Staubli VAL3: IO.pjx

--- IO.pjx ---
Parameters version=s7.7 stackSize=5000 millimeterUnit=true
Program file=Action.pgx
Program file=ActionLCF.pgx
Program file=Alarm.pgx
Program file=AtHome.pgx
Program file=AtHomePulse.pgx
Program file=Axis7Action.pgx
Program file=Axis7onPosition.pgx
Program file=Axis7OnReady.pgx
Program file=Axis7Status.pgx
Program file=Axis8Action.pgx
Program file=Axis8onPosition.pgx
Program file=Axis8OnReady.pgx
Program file=Axis8Status.pgx
Program file=AxisDoor.pgx
Program file=AxisIsNeg.pgx
Program file=AxisJogSpeed.pgx
Program file=AxisTest.pgx
Program file=CanProduct.pgx
Program file=ChoosehansPro.pgx
Program file=ChooseMultPro.pgx
Program file=CloseWeld.pgx
Program file=Digtal2Analog.pgx
Program file=Digtal2AnalogS.pgx
Program file=ExtraContrAxis.pgx
Program file=GasChoose.pgx
Program file=GetAxis7Pos.pgx
Program file=GetAxis8Pos.pgx
Program file=GetAxisStatus.pgx
Program file=GetKeyIO.pgx
Program file=GetPreset.pgx
Program file=Init.pgx
Program file=IOName.pgx
Program file=IOvalue.pgx
Program file=IsDigtal.pgx
Program file=IsInput.pgx
Program file=KeyDigtalIO.pgx
Program file=Light.pgx
Program file=MatchSpdPreset.pgx
Program file=PerforatiAction.pgx
Program file=Preset.pgx
Program file=PresetLaser.pgx
Program file=ProductPoll.pgx
Program file=ProductReady.pgx
Program file=ReadMe.pgx
Program file=SafteyIO.pgx
Program file=SendSpeed.pgx
Program file=start.pgx
Program file=stop.pgx
Program file=TrajBypass.pgx
Program file=WaitProIOEnd.pgx
Program file=WeldAction.pgx
Program file=WeldProgChoose.pgx
Program file=WorkPlaceFinish.pgx
Data file=IO.dtx

--- IO.dtx ---
public aio aAio{}
  [In4_a7CurPosH] = {link=ModbusSrv-0\Modbus-Word\In4_a7CurPosH}
  [In4_a7CurPosL] = {link=ModbusSrv-0\Modbus-Word\In4_a7CurPosL}
  [In4_a8CurPosH] = {link=ModbusSrv-0\Modbus-Word\In4_a8CurPosH}
  [In4_a8CurPosL] = {link=ModbusSrv-0\Modbus-Word\In4_a8CurPosL}
  [In_aVersion] = {link=ModbusSrv-0\Modbus-Word\In_aVersion}
  [O1_aAirPress] = {link=ModbusSrv-0\Modbus-Word\O1_aAirPress}
  [O1_aFPWM] = {link=ModbusSrv-0\Modbus-Word\O1_aFPWM}
  [O1_aLasPwr] = {link=ModbusSrv-0\Modbus-Word\O1_aLasPwr}
  [O1_aPMW] = {link=ModbusSrv-0\Modbus-Word\O1_aPMW}
  [O2_aFollowSensitive] = {link=ModbusSrv-0\Modbus-Word\O2_aFollowSensitive}
  [O2_aNull] = {link=ModbusSrv-0\Modbus-Word\O2_aNull}
  [O4_a7AiHomeH] = {link=ModbusSrv-0\Modbus-Word\O4_a7AiHomeH}
  [O4_a7AiHomeL] = {link=ModbusSrv-0\Modbus-Word\O4_a7AiHomeL}
  [O4_a7JogVelo] = {link=ModbusSrv-0\Modbus-Word\O4_a7JogVelo}
  [O4_a7MoveDis] = {link=ModbusSrv-0\Modbus-Word\O4_a7MoveDis}
  [O4_a7MovePosH] = {link=ModbusSrv-0\Modbus-Word\O4_a7MovePosH}
  [O4_a7MovePosL] = {link=ModbusSrv-0\Modbus-Word\O4_a7MovePosL}
  [O4_a7Velocity] = {link=ModbusSrv-0\Modbus-Word\O4_a7Velocity}
  [O4_a8AiHomeH] = {link=ModbusSrv-0\Modbus-Word\O4_a8AiHomeH}
  [O4_a8AiHomeL] = {link=ModbusSrv-0\Modbus-Word\O4_a8AiHomeL}
  [O4_a8JogVelo] = {link=ModbusSrv-0\Modbus-Word\O4_a8JogVelo}
  [O4_a8MoveDis] = {link=ModbusSrv-0\Modbus-Word\O4_a8MoveDis}
  [O4_a8MovePosH] = {link=ModbusSrv-0\Modbus-Word\O4_a8MovePosH}
  [O4_a8MovePosL] = {link=ModbusSrv-0\Modbus-Word\O4_a8MovePosL}
  [O4_a8Velocity] = {link=ModbusSrv-0\Modbus-Word\O4_a8Velocity}
  [Out_a114_129] = {link=ModbusSrv-0\Modbus-Word\Out_a114_129}
  [Out_a130_133] = {link=ModbusSrv-0\Modbus-Word\Out_a130_133}
  [Out_a66_81] = {link=ModbusSrv-0\Modbus-Word\Out_a66_81}
  [Out_a82_97] = {link=ModbusSrv-0\Modbus-Word\Out_a82_97}
  [Out_a98_113] = {link=ModbusSrv-0\Modbus-Word\Out_a98_113}
public bool bAxisDoorEnable
bool bDigFollowHight
public bool bDigtal[167]
  [0] = true
  [1] = true
  [2] = true
  [3] = true
  [4] = true
  [5] = true
  [6] = true
  [7] = true
  [8] = true
  [9] = true
  [10] = true
  [11] = true
  [12] = true
  [13] = true
  [14] = true
  [15] = true
  [16] = true
  [17] = true
  [18] = true
  [19] = true
  [20] = true
  [21] = true
  [22] = true
  [23] = true
  [24] = true
  [25] = true
  [26] = true
  [27] = true
  [28] = true
  [29] = true
  [30] = true
  [31] = true
  [32] = true
  [33] = true
  [34] = true
  [35] = true
  [36] = true
  [37] = true
  [38] = true
  [39] = true
  [40] = true
  [41] = true
  [42] = true
  [43] = true
  [44] = true
  [45] = true
  [46] = true
  [47] = true
  [48] = true
  [49] = true
  [50] = true
  [51] = true
  [52] = true
  [53] = true
  [54] = true
  [55] = true
  [56] = true
  [57] = true
  [58] = true
  [59] = true
  [60] = true
  [61] = true
  [62] = true
  [63] = true
  [64] = true
  [65] = true
  [66] = true
  [67] = true
  [68] = true
  [69] = true
  [70] = true
  [71] = true
  [72] = true
  [73] = true
  [74] = true
  [75] = true
  [76] = true
  [77] = true
  [78] = true
  [79] = true
  [80] = true
  [81] = true
  [82] = true
  [83] = true
  [84] = true
  [85] = true
  [86] = true
  [87] = true
  [88] = true
  [89] = true
  [90] = true
  [91] = true
  [92] = true
  [93] = true
  [94] = true
  [95] = true
  [96] = true
  [97] = true
  [98] = true
  [99] = true
  [100] = true
  [101] = true
  [102] = true
  [103] = true
  [104] = true
  [105] = true
  [106] = true
  [107] = true
  [108] = true
  [109] = true
  [110] = true
  [111] = true
  [112] = true
  [113] = true
  [114] = true
  [115] = true
  [116] = true
  [117] = true
  [118] = true
  [119] = true
  [120] = true
  [121] = true
  [122] = true
  [123] = true
  [124] = true
  [125] = true
  [126] = true
  [127] = true
  [128] = true
  [129] = true
  [130] = true
  [131] = true
  [132] = true
  [133] = true
  [134] = true
public bool bExt7AxisEnable
public bool bExt8AxisEnable
public bool bGunUp
bool bWaitActionOff
bool bWaitFollowDown
public bool bWeldEnable
public dio dDio{}
  [In1_bEndCycl] = {link=ModbusSrv-0\Modbus-Bit\In1_bEndCycl}
  [In1_bHome] = {link=ModbusSrv-0\Modbus-Bit\In1_bHome}
  [In1_bNull1] = {link=ModbusSrv-0\Modbus-Bit\In1_bNull1}
  [In1_bNull2] = {link=ModbusSrv-0\Modbus-Bit\In1_bNull2}
  [In1_bNull3] = {link=ModbusSrv-0\Modbus-Bit\In1_bNull3}
  [In1_bOutAlarm] = {link=ModbusSrv-0\Modbus-Bit\In1_bOutAlarm}
  [In1_bPausCycl] = {link=ModbusSrv-0\Modbus-Bit\In1_bPausCycl}
  [In1_bPeripheralReady] = {link=ModbusSrv-0\Modbus-Bit\In1_bPeripheralReady}
  [In1_bPowerOn] = {link=ModbusSrv-0\Modbus-Bit\In1_bPowerOn}
  [In1_bPrdSta1] = {link=ModbusSrv-0\Modbus-Bit\In1_bPrdSta1}
  [In1_bPrdSta2] = {link=ModbusSrv-0\Modbus-Bit\In1_bPrdSta2}
  [In1_bReset] = {link=ModbusSrv-0\Modbus-Bit\In1_bReset}
  [In1_bStartCycl] = {link=ModbusSrv-0\Modbus-Bit\In1_bStartCycl}
  [In1_bStopCycl] = {link=ModbusSrv-0\Modbus-Bit\In1_bStopCycl}
  [In2_bAirAlarm] = {link=ModbusSrv-0\Modbus-Bit\In2_bAirAlarm}
  [In2_bCollisonAlarm] = {link=ModbusSrv-0\Modbus-Bit\In2_bCollisonAlarm}
  [In2_bContactAlarm] = {link=ModbusSrv-0\Modbus-Bit\In2_bContactAlarm}
  [In2_bLaserAlarm] = {link=ModbusSrv-0\Modbus-Bit\In2_bLaserAlarm}
  [In2_bNull1] = {link=ModbusSrv-0\Modbus-Bit\In2_bNull1}
  [In2_bNull2] = {link=ModbusSrv-0\Modbus-Bit\In2_bNull2}
  [In2_bNull3] = {link=ModbusSrv-0\Modbus-Bit\In2_bNull3}
  [In2_bNull4] = {link=ModbusSrv-0\Modbus-Bit\In2_bNull4}
  [In2_bNull5] = {link=ModbusSrv-0\Modbus-Bit\In2_bNull5}
  [In2_bNull6] = {link=ModbusSrv-0\Modbus-Bit\In2_bNull6}
  [In2_bNull7] = {link=ModbusSrv-0\Modbus-Bit\In2_bNull7}
  [In2_bNull8] = {link=ModbusSrv-0\Modbus-Bit\In2_bNull8}
  [In2_bNull9] = {link=ModbusSrv-0\Modbus-Bit\In2_bNull9}
  [In2_bPrdSta3] = {link=ModbusSrv-0\Modbus-Bit\In2_bPrdSta3}
  [In2_bPrdSta4] = {link=ModbusSrv-0\Modbus-Bit\In2_bPrdSta4}
  [In2_bRasterOn] = {link=ModbusSrv-0\Modbus-Bit\In2_bRasterOn}
  [In4_b7BackHome] = {link=ModbusSrv-0\Modbus-Bit\In4_b7BackHome}
  [In4_b7HomeDone] = {link=ModbusSrv-0\Modbus-Bit\In4_b7HomeDone}
  [In4_b7IsHome] = {link=ModbusSrv-0\Modbus-Bit\In4_b7IsHome}
  [In4_b7MotorError] = {link=ModbusSrv-0\Modbus-Bit\In4_b7MotorError}
  [In4_b7MotorPower] = {link=ModbusSrv-0\Modbus-Bit\In4_b7MotorPower}
  [In4_b7Reached] = {link=ModbusSrv-0\Modbus-Bit\In4_b7Reached}
  [In4_b8BackHome] = {link=ModbusSrv-0\Modbus-Bit\In4_b8BackHome}
  [In4_b8HomeDone] = {link=ModbusSrv-0\Modbus-Bit\In4_b8HomeDone}
  [In4_b8IsHome] = {link=ModbusSrv-0\Modbus-Bit\In4_b8IsHome}
  [In4_b8MotorError] = {link=ModbusSrv-0\Modbus-Bit\In4_b8MotorError}
  [In4_b8MotorPower] = {link=ModbusSrv-0\Modbus-Bit\In4_b8MotorPower}
  [In4_b8Reached] = {link=ModbusSrv-0\Modbus-Bit\In4_b8Reached}
  [In4_bNull1] = {link=ModbusSrv-0\Modbus-Bit\In4_bNull1}
  [In4_bNull2] = {link=ModbusSrv-0\Modbus-Bit\In4_bNull2}
  [In4_bNull3] = {link=ModbusSrv-0\Modbus-Bit\In4_bNull3}
  [In4_bNull4] = {link=ModbusSrv-0\Modbus-Bit\In4_bNull4}
  [In4_bNull5] = {link=ModbusSrv-0\Modbus-Bit\In4_bNull5}
  [In4_bNull6] = {link=ModbusSrv-0\Modbus-Bit\In4_bNull6}
  [In4_bNull7] = {link=ModbusSrv-0\Modbus-Bit\In4_bNull7}
  [In4_bNull8] = {link=ModbusSrv-0\Modbus-Bit\In4_bNull8}
  [In7_bDownLimit_7] = {link=ModbusSrv-0\Modbus-Bit\In7_bDownLimit_7}
  [In7_bHomeLimit_7] = {link=ModbusSrv-0\Modbus-Bit\In7_bHomeLimit_7}
  [In7_bNull1] = {link=ModbusSrv-0\Modbus-Bit\In7_bNull1}
  [In7_bUpLimit_7] = {link=ModbusSrv-0\Modbus-Bit\In7_bUpLimit_7}
  [In8_bDownLimit_8] = {link=ModbusSrv-0\Modbus-Bit\In8_bDownLimit_8}
  [In8_bHomeLimit_8] = {link=ModbusSrv-0\Modbus-Bit\In8_bHomeLimit_8}
  [In8_bNull1] = {link=ModbusSrv-0\Modbus-Bit\In8_bNull1}
  [In8_bUpLimit_8] = {link=ModbusSrv-0\Modbus-Bit\In8_bUpLimit_8}
  [O1_bAirOn] = {link=ModbusSrv-0\Modbus-Bit\O1_bAirOn}
  [O1_bAlarm] = {link=ModbusSrv-0\Modbus-Bit\O1_bAlarm}
  [O1_bFollowDone] = {link=ModbusSrv-0\Modbus-Bit\O1_bFollowDone}
  [O1_bFollowOn] = {link=ModbusSrv-0\Modbus-Bit\O1_bFollowOn}
  [O1_bGreenLamp] = {link=ModbusSrv-0\Modbus-Bit\O1_bGreenLamp}
  [O1_bLaserOn] = {link=ModbusSrv-0\Modbus-Bit\O1_bLaserOn}
  [O1_bNull1] = {link=ModbusSrv-0\Modbus-Bit\O1_bNull1}
  [O1_bRedLamp] = {link=ModbusSrv-0\Modbus-Bit\O1_bRedLamp}
  [O1_bYellowLamp] = {link=ModbusSrv-0\Modbus-Bit\O1_bYellowLamp}
  [O2_bAxisPos1] = {link=ModbusSrv-0\Modbus-Bit\O2_bAxisPos1}
  [O2_bAxisPos2] = {link=ModbusSrv-0\Modbus-Bit\O2_bAxisPos2}
  [O2_bAxisPos3] = {link=ModbusSrv-0\Modbus-Bit\O2_bAxisPos3}
  [O2_bFollowHeigh1] = {link=ModbusSrv-0\Modbus-Bit\O2_bFollowHeigh1}
  [O2_bFollowHeigh2] = {link=ModbusSrv-0\Modbus-Bit\O2_bFollowHeigh2}
  [O2_bFollowHeigh3] = {link=ModbusSrv-0\Modbus-Bit\O2_bFollowHeigh3}
  [O2_bNull1] = {link=ModbusSrv-0\Modbus-Bit\O2_bNull1}
  [O2_bNull2] = {link=ModbusSrv-0\Modbus-Bit\O2_bNull2}
  [O2_bNull3] = {link=ModbusSrv-0\Modbus-Bit\O2_bNull3}
  [O2_bProCode1] = {link=ModbusSrv-0\Modbus-Bit\O2_bProCode1}
  [O2_bProCode2] = {link=ModbusSrv-0\Modbus-Bit\O2_bProCode2}
  [O2_bProCode3] = {link=ModbusSrv-0\Modbus-Bit\O2_bProCode3}
  [O2_bSta1Stat] = {link=ModbusSrv-0\Modbus-Bit\O2_bSta1Stat}
  [O2_bSta2Stat] = {link=ModbusSrv-0\Modbus-Bit\O2_bSta2Stat}
  [O2_bSta3Stat] = {link=ModbusSrv-0\Modbus-Bit\O2_bSta3Stat}
  [O2_bSta4Stat] = {link=ModbusSrv-0\Modbus-Bit\O2_bSta4Stat}
  [O4_b7AxisHome] = {link=ModbusSrv-0\Modbus-Bit\O4_b7AxisHome}
  [O4_b7ChkHome] = {link=ModbusSrv-0\Modbus-Bit\O4_b7ChkHome}
  [O4_b7MoveDir] = {link=ModbusSrv-0\Modbus-Bit\O4_b7MoveDir}
  [O4_b7MoveDirM] = {link=ModbusSrv-0\Modbus-Bit\O4_b7MoveDirM}
  [O4_b7MoveToPos] = {link=ModbusSrv-0\Modbus-Bit\O4_b7MoveToPos}
  [O4_b7RecordPos] = {link=ModbusSrv-0\Modbus-Bit\O4_b7RecordPos}
  [O4_b7ResetError] = {link=ModbusSrv-0\Modbus-Bit\O4_b7ResetError}
  [O4_b7StopMotor] = {link=ModbusSrv-0\Modbus-Bit\O4_b7StopMotor}
  [O4_b8AxisHome] = {link=ModbusSrv-0\Modbus-Bit\O4_b8AxisHome}
  [O4_b8ChkHome] = {link=ModbusSrv-0\Modbus-Bit\O4_b8ChkHome}
  [O4_b8MoveDir] = {link=ModbusSrv-0\Modbus-Bit\O4_b8MoveDir}
  [O4_b8MoveDirM] = {link=ModbusSrv-0\Modbus-Bit\O4_b8MoveDirM}
  [O4_b8MoveToPos] = {link=ModbusSrv-0\Modbus-Bit\O4_b8MoveToPos}
  [O4_b8RecordPos] = {link=ModbusSrv-0\Modbus-Bit\O4_b8RecordPos}
  [O4_b8ResetError] = {link=ModbusSrv-0\Modbus-Bit\O4_b8ResetError}
  [O4_b8StopMotor] = {link=ModbusSrv-0\Modbus-Bit\O4_b8StopMotor}
  [O4_bHome] = {link=ModbusSrv-0\Modbus-Bit\O4_bHome}
  [O4_bNull1] = {link=ModbusSrv-0\Modbus-Bit\O4_bNull1}
  [O4_bNull2] = {link=ModbusSrv-0\Modbus-Bit\O4_bNull2}
  [O4_bNull3] = {link=ModbusSrv-0\Modbus-Bit\O4_bNull3}
  [O4_bNull4] = {link=ModbusSrv-0\Modbus-Bit\O4_bNull4}
  [O4_bNull5] = {link=ModbusSrv-0\Modbus-Bit\O4_bNull5}
  [O4_bNull6] = {link=ModbusSrv-0\Modbus-Bit\O4_bNull6}
  [O4_bNull7] = {link=ModbusSrv-0\Modbus-Bit\O4_bNull7}
  [O4_bNull8] = {link=ModbusSrv-0\Modbus-Bit\O4_bNull8}
  [O7_bAxis7Direction] = {link=ModbusSrv-0\Modbus-Bit\O7_bAxis7Direction}
  [O7_bAxis7Pulse] = {link=ModbusSrv-0\Modbus-Bit\O7_bAxis7Pulse}
  [O7_bNull1] = {link=ModbusSrv-0\Modbus-Bit\O7_bNull1}
  [O7_bNull2] = {link=ModbusSrv-0\Modbus-Bit\O7_bNull2}
  [O7_bNull3] = {link=ModbusSrv-0\Modbus-Bit\O7_bNull3}
  [O8_bAxis8Direction] = {link=ModbusSrv-0\Modbus-Bit\O8_bAxis8Direction}
  [O8_bAxis8Pulse] = {link=ModbusSrv-0\Modbus-Bit\O8_bAxis8Pulse}
  [O8_bNull1] = {link=ModbusSrv-0\Modbus-Bit\O8_bNull1}
  [O8_bNull2] = {link=ModbusSrv-0\Modbus-Bit\O8_bNull2}
  [O8_bNull3] = {link=ModbusSrv-0\Modbus-Bit\O8_bNull3}
  [UsIn_bNull1] = {link=ModbusSrv-0\Modbus-Bit\UsIn_bNull1}
  [UsIn_bNull2] = {link=ModbusSrv-0\Modbus-Bit\UsIn_bNull2}
  [UsIn_bNull3] = {link=ModbusSrv-0\Modbus-Bit\UsIn_bNull3}
  [UsIn_bNull4] = {link=ModbusSrv-0\Modbus-Bit\UsIn_bNull4}
  [UsIn_bNull5] = {link=ModbusSrv-0\Modbus-Bit\UsIn_bNull5}
  [UsIn_bNull6] = {link=ModbusSrv-0\Modbus-Bit\UsIn_bNull6}
  [UsIn_bNull7] = {link=ModbusSrv-0\Modbus-Bit\UsIn_bNull7}
  [UsIn_bNull8] = {link=ModbusSrv-0\Modbus-Bit\UsIn_bNull8}
  [UsO_bNull1] = {link=ModbusSrv-0\Modbus-Bit\UsO_bNull1}
  [UsO_bNull2] = {link=ModbusSrv-0\Modbus-Bit\UsO_bNull2}
  [UsO_bNull3] = {link=ModbusSrv-0\Modbus-Bit\UsO_bNull3}
  [UsO_bNull4] = {link=ModbusSrv-0\Modbus-Bit\UsO_bNull4}
  [UsO_bNull5] = {link=ModbusSrv-0\Modbus-Bit\UsO_bNull5}
  [UsO_bNull6] = {link=ModbusSrv-0\Modbus-Bit\UsO_bNull6}
  [UsO_bNull7] = {link=ModbusSrv-0\Modbus-Bit\UsO_bNull7}
  [UsO_bNull8] = {link=ModbusSrv-0\Modbus-Bit\UsO_bNull8}
public string sIOName[167]
  [0] = "无"
  [1] = "In1_bPowerOn"
  [2] = "In1_bStartCycl"
  [3] = "In1_bStopCycl"
  [4] = "In1_bHome"
  [5] = "In1_bEndCycl"
  [6] = "In1_bPrdSta1"
  [7] = "In1_bPrdSta2"
  [8] = "In1_bPausCycl"
  [9] = "In1_bOutAlarm"
  [10] = "In1_bReset"
  [11] = "In1_bPeripheralReady"
  [12] = "In1_bNull1"
  [13] = "In1_bNull2"
  [14] = "In1_bNull3"
  [15] = "UsIn_bNull1"
  [16] = "UsIn_bNull2"
  [17] = "UsIn_bNull3"
  [18] = "UsIn_bNull4"
  [19] = "UsIn_bNull5"
  [20] = "UsIn_bNull6"
  [21] = "UsIn_bNull7"
  [22] = "UsIn_bNull8"
  [23] = "In2_bPrdSta3"
  [24] = "In2_bPrdSta4"
  [25] = "In2_bAirAlarm"
  [26] = "In2_bCollisonAlarm"
  [27] = "In2_bLaserAlarm"
  [28] = "In2_bContactAlarm"
  [29] = "In2_bRasterOn"
  [30] = "In2_bNull1"
  [31] = "In2_bNull2"
  [32] = "In2_bNull3"
  [33] = "In2_bNull4"
  [34] = "In2_bNull5"
  [35] = "In2_bNull6"
  [36] = "In2_bNull7"
  [37] = "In2_bNull8"
  [38] = "In2_bNull9"
  [39] = "In7_bUpLimit_7"
  [40] = "In7_bDownLimit_7"
  [41] = "In7_bHomeLimit_7"
  [42] = "In7_bNull1"
  [43] = "In8_bUpLimit_8"
  [44] = "In8_bDownLimit_8"
  [45] = "In8_bHomeLimit_8"
  [46] = "In8_bNull1"
  [47] = "In4_b7Reached"
  [48] = "In4_b7BackHome"
  [49] = "In4_b7HomeDone"
  [50] = "In4_b7MotorPower"
  [51] = "In4_b7IsHome"
  [52] = "In4_b7MotorError"
  [53] = "In4_b8Reached"
  [54] = "In4_b8BackHome"
  [55] = "In4_b8HomeDone"
  [56] = "In4_b8MotorPower"
  [57] = "In4_b8IsHome"
  [58] = "In4_b8MotorError"
  [59] = "In4_bNull1"
  [60] = "In4_bNull2"
  [61] = "In4_bNull3"
  [62] = "In4_bNull4"
  [63] = "In4_bNull5"
  [64] = "In4_bNull6"
  [65] = "In4_bNull7"
  [66] = "In4_bNull8"
  [67] = "O1_bLaserOn"
  [68] = "O1_bFollowOn"
  [69] = "O1_bFollowDone"
  [70] = "O1_bAirOn"
  [71] = "O1_bNull1"
  [72] = "O1_bRedLamp"
  [73] = "O1_bYellowLamp"
  [74] = "O1_bGreenLamp"
  [75] = "O1_bAlarm"
  [76] = "UsO_bNull1"
  [77] = "UsO_bNull2"
  [78] = "UsO_bNull3"
  [79] = "UsO_bNull4"
  [80] = "UsO_bNull5"
  [81] = "UsO_bNull6"
  [82] = "UsO_bNull7"
  [83] = "UsO_bNull8"
  [84] = "O2_bSta1Stat"
  [85] = "O2_bSta2Stat"
  [86] = "O2_bSta3Stat"
  [87] = "O2_bSta4Stat"
  [88] = "O2_bProCode1"
  [89] = "O2_bProCode2"
  [90] = "O2_bProCode3"
  [91] = "O2_bFollowHeigh1"
  [92] = "O2_bFollowHeigh2"
  [93] = "O2_bFollowHeigh3"
  [94] = "O2_bAxisPos1"
  [95] = "O2_bAxisPos2"
  [96] = "O2_bAxisPos3"
  [97] = "O2_bNull1"
  [98] = "O2_bNull2"
  [99] = "O2_bNull3"
  [100] = "O7_bAxis7Pulse"
  [101] = "O7_bAxis7Direction"
  [102] = "O7_bNull1"
  [103] = "O7_bNull2"
  [104] = "O7_bNull3"
  [105] = "O8_bAxis8Pulse"
  [106] = "O8_bAxis8Direction"
  [107] = "O8_bNull1"
  [108] = "O8_bNull2"
  [109] = "O8_bNull3"
  [110] = "O4_b7RecordPos"
  [111] = "O4_b7MoveToPos"
  [112] = "O4_b7ResetError"
  [113] = "O4_b7ChkHome"
  [114] = "O4_b7AxisHome"
  [115] = "O4_b7MoveDir"
  [116] = "O4_b7MoveDirM"
  [117] = "O4_b7StopMotor"
  [118] = "O4_bHome"
  [119] = "O4_b8RecordPos"
  [120] = "O4_b8MoveToPos"
  [121] = "O4_b8ResetError"
  [122] = "O4_b8ChkHome"
  [123] = "O4_b8AxisHome"
  [124] = "O4_b8MoveDir"
  [125] = "O4_b8MoveDirM"
  [126] = "O4_b8StopMotor"
  [127] = "O4_bNull1"
  [128] = "O4_bNull2"
  [129] = "O4_bNull3"
  [130] = "O4_bNull4"
  [131] = "O4_bNull5"
  [132] = "O4_bNull6"
  [133] = "O4_bNull7"
  [134] = "O4_bNull8"
  [135] = "O1_aLasPwr"
  [136] = "O1_aAirPress"
  [137] = "O1_aFPWM"
  [138] = "O1_aPMW"
  [139] = "O2_aFollowSensitive"
  [140] = "O2_aNull"
  [141] = "In4_a7CurPosL"
  [142] = "In4_a7CurPosH"
  [143] = "In4_a8CurPosL"
  [144] = "In4_a8CurPosH"
  [145] = "O4_a7Velocity"
  [146] = "O4_a7JogVelo"
  [147] = "O4_a7MoveDis"
  [148] = "O4_a7AiHomeH"
  [149] = "O4_a7AiHomeL"
  [150] = "O4_a7MovePosL"
  [151] = "O4_a7MovePosH"
  [152] = "O4_a8Velocity"
  [153] = "O4_a8JogVelo"
  [154] = "O4_a8MoveDis"
  [155] = "O4_a8AiHomeH"
  [156] = "O4_a8AiHomeL"
  [157] = "O4_a8MovePosL"
  [158] = "O4_a8MovePosH"
  [159] = "Out_a66_81"
  [160] = "Out_a82_97"
  [161] = "Out_a98_113"
  [162] = "Out_a114_129"
  [163] = "Out_a130_133"
  [164] = "In_aVersion"
  [165] = "延时"
  [166] = "收弧时间"
public bool bUserIOReset

--- IO123.dtx ---
mdesc mNomSpeed
public string sIOName
public bool bDigtal

--- start.pgx ---
public program start()
begin
  //所有的IO动作都要写入log文件中
  //信号一般作为脉冲信号来处理
  //



  call Init()

  while true


    call Digtal2Analog()
    delay(0)
  endWhile
end

--- Action.pgx ---
public program Action(num& x_nAction[] (dimensions=2), bool x_bMoveId, num x_nMoveID)
  local bool l_bFirst
  local bool l_bInput
  local bool l_bNull
  local num l_nLast
  local num l_nNum
begin
  //延时是否需要停止等待？
  //




  //一共是每个点上最多12个IO


  //如果都为空，则直接跳出
  l_bNull=false
  for l_nNum=0 to 11
    l_bNull=x_nAction[l_nNum,0]!=0 or x_nAction[l_nNum,1]!=0 or l_bNull
  endFor
  if !l_bNull
    return
  endIf




  //通过MOVEID来实现
  for l_nNum=0 to 11

    //如果后面的都是0则退出
    l_bNull=false
    for l_nLast=l_nNum to 11
      l_bNull=x_nAction[l_nLast,0]!=0 or x_nAction[l_nLast,1]!=0 or l_bNull
    endFor
    if !l_bNull
      return
    endIf


    //通过MOVEID来实现
    if x_bMoveId
      call IsInput(x_nAction[l_nNum,0],l_bInput)
      //如果有等待信号，直接退出
      if l_bInput
        return
      else
        wait(getMoveId()>x_nMoveID+0.8)
        call IOvalue(x_nAction[l_nNum,0],x_nAction[l_nNum,1])
      endIf





     //
    else

      //跟在运动指令后面
      call IsInput(x_nAction[l_nNum,0],l_bInput)
      //如果有等待信号 则运行
      if l_bInput
        l_bFirst=true

      endIf

      if l_bFirst
        //如果不是收弧时间


        if x_nAction[l_nNum,0]!=166 and l_bInput
          if x_nMoveID==-2
            waitEndMove()
          else
            if x_nMoveID>=0
              wait(getMoveId()>x_nMoveID+0.8)
            endIf
          endIf
        endIf
      endIf

      call IOvalue(x_nAction[l_nNum,0],x_nAction[l_nNum,1])


      if x_nAction[l_nNum,0]==166
        //  logMsg(toString(".3",x_nAction[l_nNum,1]))
        logMsg(toString(".3",clock())+"  "+toString(".3",getMoveId()))
      endIf


    endIf


    //把数字量输出
    call Digtal2Analog()

  endFor


end

--- ActionLCF.pgx ---
public program ActionLCF(num& x_nAction[] (dimensions=2), bool x_bMoveId, num x_nMoveID, num x_nActionBuff)
  local bool l_bFirst
  local bool l_bInput
  local bool l_bNull
  local num l_nLast
  local num l_nNum
begin
  //2016.01.26
  //特定为激光融覆定制的程序



  //延时是否需要停止等待？
  //

  x_nActionBuff=max(0.01,min(0.8,x_nActionBuff))


  //一共是每个点上最多12个IO


  //如果都为空，则直接跳出
  l_bNull=false
  for l_nNum=0 to 11
    l_bNull=x_nAction[l_nNum,0]!=0 or x_nAction[l_nNum,1]!=0 or l_bNull
  endFor
  if !l_bNull
    return
  endIf




  //通过MOVEID来实现
  for l_nNum=0 to 11

    //如果后面的都是0则退出
    l_bNull=false
    for l_nLast=l_nNum to 11
      l_bNull=x_nAction[l_nLast,0]!=0 or x_nAction[l_nLast,1]!=0 or l_bNull
    endFor
    if !l_bNull
      return
    endIf


    //通过MOVEID来实现
    if x_bMoveId
      call IsInput(x_nAction[l_nNum,0],l_bInput)
      //如果有等待信号，直接退出
      if l_bInput
        return
      else
        wait(getMoveId()>x_nMoveID+x_nActionBuff)
        call IOvalue(x_nAction[l_nNum,0],x_nAction[l_nNum,1])
      endIf





     //
    else

      //跟在运动指令后面
      call IsInput(x_nAction[l_nNum,0],l_bInput)
      //如果有等待信号 则运行
      if l_bInput
        l_bFirst=true

      endIf

      if l_bFirst
        //如果不是收弧时间


        if x_nAction[l_nNum,0]!=166 and l_bInput
          if x_nMoveID==-2
            waitEndMove()
          else
            if x_nMoveID>=0
              wait(getMoveId()>x_nMoveID+x_nActionBuff)
            endIf
          endIf
        endIf
      endIf

      call IOvalue(x_nAction[l_nNum,0],x_nAction[l_nNum,1])


      if x_nAction[l_nNum,0]==166
        //  logMsg(toString(".3",x_nAction[l_nNum,1]))
        logMsg(toString(".3",clock())+"  "+toString(".3",getMoveId()))
      endIf


    endIf


    //把数字量输出
    call Digtal2Analog()

  endFor


end

--- Alarm.pgx ---
public program Alarm(num x_nDelay (dimensions=1), num x_nInterface (dimensions=1), bool& x_bAlarm (dimensions=1))
  local bool l_bEstop
  local string l_sS
begin
  //外设报警信号触发

  //外部綜合报警，七轴报警，八轴报警
  //碰撞报警，气体报警，随动报警


  x_bAlarm=false
  call IOName(9,l_sS)
  x_bAlarm=(x_bAlarm or dDio[l_sS]==true)
  call IOName(25,l_sS)
  x_bAlarm=(x_bAlarm or dDio[l_sS]==true)
  call IOName(26,l_sS)
  x_bAlarm=(x_bAlarm or dDio[l_sS]==true)
  call IOName(27,l_sS)
  x_bAlarm=(x_bAlarm or dDio[l_sS]==true)
  call IOName(28,l_sS)
  x_bAlarm=(x_bAlarm or dDio[l_sS]==true)

  //外部七轴报警
  if bExt7AxisEnable
    call IOName(52,l_sS)
    x_bAlarm=(x_bAlarm or dDio[l_sS]==true)
  endIf

  //外部八轴报警
  if bExt8AxisEnable
    call IOName(58,l_sS)
    x_bAlarm=(x_bAlarm or dDio[l_sS]==true)
  endIf

  delay(0)
  //急停按钮输入
  l_bEstop=esStatus()==2
  dDio["O1_bAlarm"]=l_bEstop
  x_bAlarm=(l_bEstop or x_bAlarm)

  //报警或者机器人没有上电，则会停止外部轴运动
  if x_bAlarm or !isPowered()
    if dDio["O4_b7StopMotor"]==false
      dDio["O4_b7StopMotor"]=true
    endIf
    if dDio["O4_b8StopMotor"]==false
      dDio["O4_b8StopMotor"]=true
    endIf
  endIf


  //如果再次确认报警
  if x_bAlarm

    //如果机器人在上电状态，再次确认
    if isPowered()
      delay(min(max(0,x_nDelay),5))
      //再次确认
      x_bAlarm=false
      call IOName(9,l_sS)
      x_bAlarm=(dDio[l_sS]==true or x_bAlarm)
      call IOName(25,l_sS)
      x_bAlarm=(dDio[l_sS]==true or x_bAlarm)
      call IOName(26,l_sS)
      x_bAlarm=(dDio[l_sS]==true or x_bAlarm)
      call IOName(27,l_sS)
      x_bAlarm=(dDio[l_sS]==true or x_bAlarm)
      call IOName(28,l_sS)
      x_bAlarm=(dDio[l_sS]==true or x_bAlarm)

      //外部七轴
      if bExt7AxisEnable
        call IOName(52,l_sS)
        x_bAlarm=(dDio[l_sS]==true or x_bAlarm)
      endIf

      //外部八轴
      if bExt8AxisEnable
        call IOName(58,l_sS)
        x_bAlarm=(dDio[l_sS]==true or x_bAlarm)
      endIf

    endIf

    //查看机器人是否报警
    if x_bAlarm
      call Light(0)
      if isPowered()
        disablePower()
        //        logMsg("Modbus IO输入报警触发")
        call IOName(9,l_sS)
        if dDio[l_sS]==true
          popUpMsg("In1_bOutAlarm  外部综合报警触发")
          logMsg("In1_bOutAlarm  外部综合报警触发")
        endIf


        call IOName(25,l_sS)
        if dDio[l_sS]==true
          popUpMsg("In2_bAirAlarm  气体报警触发")
          logMsg("In2_bAirAlarm  气体报警触发")
        endIf

        call IOName(26,l_sS)
        if dDio[l_sS]==true
          popUpMsg("In2_bCollisonAlarm  碰撞报警触发")
          logMsg("In2_bCollisonAlarm  碰撞报警触发")
        endIf

        call IOName(27,l_sS)
        if dDio[l_sS]==true
          popUpMsg("In2_bLaserAlarm  激光报警触发")
          logMsg("In2_bLaserAlarm  激光报警触发")
        endIf

        call IOName(28,l_sS)
        if dDio[l_sS]==true
          popUpMsg("In2_bContactAlarm  触碰报警触发")
          logMsg("In2_bContactAlarm  触碰报警触发")
        endIf

        call IOName(52,l_sS)
        if dDio[l_sS]==true
          popUpMsg("In4_b7MotorError 七轴报警触发")
          logMsg("In4_b7MotorError 七轴报警触发")
        endIf

        call IOName(58,l_sS)
        if dDio[l_sS]==true
          popUpMsg("In4_b8MotorError  八轴报警触发")
          logMsg("In4_b8MotorError  八轴报警触发")
        endIf

      endIf
      call KeyDigtalIO(false,false,false,0,0)
      //      call SafteyIO(false)
      //      call SafteyIO(true)
    endIf

  else
    if x_nInterface!=13
      call Light(1)
    endIf
  endIf

end

--- AtHome.pgx ---
public program AtHome(bool x_bHome (dimensions=1))
begin


  dDio["O1_bFollowDone"]=x_bHome
  call Digtal2Analog()







end

--- AtHomePulse.pgx ---
public program AtHomePulse()
begin

  //2014.12.09
  //回零脉冲
  waitEndMove()
  dDio["UsO_bNull2"]=true
  call Digtal2Analog()
  delay(0.5)
  dDio["UsO_bNull2"]=false
  call Digtal2Analog()


  //信号确认
  delay(0.5)
  dDio["UsO_bNull1"]=true
  delay(0.5)
  dDio["UsO_bNull1"]=false
  delay(0.5)
  dDio["UsO_bNull7"]=true
  delay(0.5)
  dDio["UsO_bNull7"]=false
  delay(0.5)


end

--- Axis7Action.pgx ---
public program Axis7Action(num x_nType (dimensions=1))
begin

  //七轴的IO动作

  switch x_nType

    //点动正
    case 1
      if dDio["O4_b7StopMotor"]==true
        dDio["O4_b7StopMotor"]=false
        delay(0.05)
      endIf
      dDio["O4_b7MoveDir"]=true
      // aioSet(aAio["O4_a7JogVelo"],50)
      delay(0.2)

    break


    //点动负
    case 2
      if dDio["O4_b7StopMotor"]==true
        dDio["O4_b7StopMotor"]=false
        delay(0.05)
      endIf

      dDio["O4_b7MoveDirM"]=true
      //  aioSet(aAio["O4_a7JogVelo"],50)
      delay(0.2)
    break

    //回到机械零位
    case 4
      dDio["O4_b7StopMotor"]=false
      dDio["O4_b7AxisHome"]=true
      delay(0.2)
    break





    //停止运动
    case 6
      dDio["O4_b7StopMotor"]=true
      delay(0.2)
      dDio["O4_b7StopMotor"]=false
    break




    //没有按钮按下
    case 9
      dDio["O4_b7ResetError"]=false
      dDio["O4_b7AxisHome"]=false
      dDio["O4_b7MoveDirM"]=false
      dDio["O4_b7MoveDir"]=false
    break


    //复位
    case 10
      dDio["O4_b7StopMotor"]=false
      dDio["O4_b7ResetError"]=true
      delay(0.2)
      // dDio["O4_b7ResetError"]=false
    break
    default
    break

  endSwitch


end

--- Axis7onPosition.pgx ---
public program Axis7onPosition(num x_nPos (dimensions=1), num x_nPrecent (dimensions=1), bool& x_bOK (dimensions=1))
  local num l_nNum
begin

  x_bOK=false
  call GetAxis7Pos(l_nNum,x_nPrecent)
  x_bOK=abs(l_nNum-x_nPos)<0.001

end

--- Axis7OnReady.pgx ---
public program Axis7OnReady(num x_nPosition (dimensions=1), num x_nSpeed (dimensions=1), num x_nPrecent (dimensions=1), bool& x_bRes (dimensions=1))
  local bool l_bBool
  local num l_nNum
begin

  //异步七轴运动到位


  x_bRes=false

  //参数合法性
  if x_nSpeed<=0 or x_nPrecent<=0 or x_nPosition<=0
    return
  endIf


  //没有电或者报警
  if dDio["In4_b7MotorPower"]==false or dDio["In4_b7MotorError"]==true or dDio["In4_b7BackHome"]==false
    return
  endIf

  call AxisIsNeg(false,l_bBool)
  if l_bBool
    return
  endIf


  dDio["O4_b7RecordPos"]=true
  delay(0.2)
  dDio["O4_b7RecordPos"]=false

  call GetAxis7Pos(l_nNum,x_nPrecent)
  if abs(l_nNum-x_nPosition)!=0
    waitEndMove()
  else
    x_bRes=true
    return
  endIf
  dDio["O4_b7StopMotor"]=false
  delay(0.2)
  x_nPosition=x_nPosition*x_nPrecent
  aioSet(aAio["O4_a7Velocity"],max(1,x_nSpeed*x_nPrecent*16.666667))
  aioSet(aAio["O4_a7MovePosL"],x_nPosition%power(2,16))
  aioSet(aAio["O4_a7MovePosH"],roundDown(x_nPosition/power(2,16)))
  dDio["O4_b7MoveToPos"]=true
  delay(0.2)
  dDio["O4_b7MoveToPos"]=false

  x_nPosition=x_nPosition/x_nPrecent
  while dDio["In4_b7Reached"]!=true or abs(l_nNum-x_nPosition)>10
    call GetAxis7Pos(l_nNum,x_nPrecent)
    if dDio["O4_b7StopMotor"]==true
      x_bRes=false
      return
    endIf
    delay(0)
  endWhile

  x_bRes=true



end

--- Axis7Status.pgx ---
public program Axis7Status(bool& x_bPowerOn (dimensions=1), bool& x_bAlarm (dimensions=1), bool& x_bhome (dimensions=1))
begin

  //  x_bAlarm=true
  //  x_bPowerOn=false

  x_bhome=dDio["In4_b7BackHome"]==true
  x_bPowerOn=dDio["In4_b7MotorPower"]==true
  x_bAlarm=dDio["In4_b7MotorError"]==true











end

--- Axis8Action.pgx ---
public program Axis8Action(num x_nType (dimensions=1))
begin

  //七轴的IO动作

  switch x_nType

    //点动正
    case 1
      if dDio["O4_b8StopMotor"]==true
        dDio["O4_b8StopMotor"]=false
        delay(0.05)
      endIf
      dDio["O4_b8MoveDir"]=true
      //aioSet(aAio["O4_a8JogVelo"],50)
      delay(0.2)

    break

    //点动负
    case 2
      if dDio["O4_b8StopMotor"]==true
        dDio["O4_b8StopMotor"]=false
        delay(0.05)
      endIf
      dDio["O4_b8MoveDirM"]=true
      //  aioSet(aAio["O4_a8JogVelo"],50)
      delay(0.2)
    break

    //回到机械零位
    case 4
      dDio["O4_b8StopMotor"]=false
      dDio["O4_b8AxisHome"]=true
      delay(0.2)
    break





    //停止运动
    case 6
      dDio["O4_b8StopMotor"]=true
      delay(0.2)
      dDio["O4_b8StopMotor"]=false
    break


    case 6

    break


    //没有按钮按下
    case 9
      dDio["O4_b8ResetError"]=false
      dDio["O4_b8AxisHome"]=false
      dDio["O4_b8MoveDirM"]=false
      dDio["O4_b8MoveDir"]=false
    break


    //复位
    case 10
      dDio["O4_b8StopMotor"]=false
      dDio["O4_b8ResetError"]=true
      // dDio["O4_b8StopMotor"]=false
      delay(0.2)
    break
    default
    break

  endSwitch


end

--- Axis8onPosition.pgx ---
public program Axis8onPosition(num x_nPos (dimensions=1), num x_nPrecent (dimensions=1), bool& x_bOK (dimensions=1))
  local num l_nNum
begin

  x_bOK=false
  call GetAxis8Pos(l_nNum,x_nPrecent)
  x_bOK=abs(l_nNum-x_nPos)<0.001

end

--- Axis8OnReady.pgx ---
public program Axis8OnReady(num x_nPosition (dimensions=1), num x_nSpeed (dimensions=1), num x_nPrecent (dimensions=1), bool& x_bRes (dimensions=1))
  local bool l_bBool
  local num l_nNum
begin


  //异步八轴到位
  x_bRes=false

  //参数合法性
  if x_nSpeed<=0 or x_nPrecent<=0 or x_nPosition<=0
    return
  endIf



  //没有电或者报警
  if dDio["In4_b8MotorPower"]==false or dDio["In4_b8MotorError"]==true or dDio["In4_b8BackHome"]==false
    return
  endIf

  call AxisIsNeg(true,l_bBool)
  if l_bBool
    return
  endIf


  dDio["O4_b8RecordPos"]=true
  delay(0.2)
  dDio["O4_b8RecordPos"]=false

  call GetAxis8Pos(l_nNum,x_nPrecent)

  if abs(l_nNum-x_nPosition)!=0
    waitEndMove()
  else
    x_bRes=true
    return
  endIf

  dDio["O4_b8StopMotor"]=false
  delay(0.2)
  x_nPosition=x_nPosition*x_nPrecent
  aioSet(aAio["O4_a8Velocity"],max(1,x_nSpeed*x_nPrecent*16.666667))
  aioSet(aAio["O4_a8MovePosL"],x_nPosition%power(2,16))
  aioSet(aAio["O4_a8MovePosH"],roundDown(x_nPosition/power(2,16)))
  dDio["O4_b8MoveToPos"]=true
  delay(0.2)
  dDio["O4_b8MoveToPos"]=false

  x_nPosition=x_nPosition/x_nPrecent
  while dDio["In4_b8Reached"]!=true or abs(l_nNum-x_nPosition)>10
    call GetAxis8Pos(l_nNum,x_nPrecent)
    if dDio["O4_b8StopMotor"]==true
      x_bRes=false
      return
    endIf
    delay(0)
  endWhile

  x_bRes=true


end

--- Axis8Status.pgx ---
public program Axis8Status(bool& x_bPowerOn (dimensions=1), bool& x_bAlarm (dimensions=1), bool& x_bhome (dimensions=1))
begin
  //  x_bAlarm=true
  //  x_bPowerOn=false
  x_bhome=dDio["In4_b8BackHome"]==true
  x_bPowerOn=dDio["In4_b8MotorPower"]==true
  x_bAlarm=dDio["In4_b8MotorError"]==true


end

--- AxisDoor.pgx ---
public program AxisDoor(bool x_bOpen (dimensions=1), bool x_b8Axis (dimensions=1))
begin
  //门开关信号
  //为外部轴七轴和八轴进行打开安全门使用
  //法利莱
  //安全门信号设置


  //如果门打不开，则打不开
  if !bAxisDoorEnable
    return
  endIf


  //x_bOpen   true 打开门   false 门关闭
  //x_b8Axis  true  八轴    false 七轴


  //七八轴打开
  if !x_b8Axis
    //七轴打开
    if x_bOpen
      dDio["UsO_bNull5"]=true
      wait(dDio["UsIn_bNull5"]==true and dDio["UsIn_bNull6"]==false)
    else
      dDio["UsO_bNull5"]=false
      wait(dDio["UsIn_bNull6"]==true and dDio["UsIn_bNull5"]==false)

    endIf


  else
    //八轴打开
    if x_bOpen
      dDio["UsO_bNull6"]=true
      wait(dDio["UsIn_bNull7"]==true and dDio["UsIn_bNull8"]==false)
    else
      dDio["UsO_bNull6"]=false
      wait(dDio["UsIn_bNull8"]==true and dDio["UsIn_bNull7"]==false)

    endIf
  endIf



end

--- AxisIsNeg.pgx ---
public program AxisIsNeg(bool x_b8Axis (dimensions=1), bool& x_bRes (dimensions=1))
begin
  x_bRes=false

  if x_b8Axis
    x_bRes=aioGet(aAio["In4_a8CurPosH"])>=3000

  else

    x_bRes=aioGet(aAio["In4_a7CurPosH"])>=3000

  endIf





end

--- AxisJogSpeed.pgx ---
public program AxisJogSpeed(num x_nSpeed, bool x_b8Axis)
begin

  //修改点动速度
  //修改1这个是比例系数

  x_nSpeed=max(0,min(100,x_nSpeed))
  if x_b8Axis

    aioSet(aAio["O4_a8JogVelo"],x_nSpeed*1)

  else
    aioSet(aAio["O4_a7JogVelo"],x_nSpeed*1)

  endIf




end

--- AxisTest.pgx ---
public program AxisTest()
begin
  dDio["O1_bFollowOn"]=true
  delay(0.5)
  dDio["O1_bFollowOn"]=false
  delay(0.5)
  dDio["O1_bFollowOn"]=true
  delay(0.5)
  dDio["O1_bFollowOn"]=false
  delay(0.5)


end

--- CanProduct.pgx ---
public program CanProduct(num& x_nWorkPlace (dimensions=1))
begin
  //等待IO响应



  //第一工位
  if dDio["In1_bPrdSta1"]==true
    delay(0.2)
    if watch(dDio["In1_bPrdSta1"]==true,0.1)
      if watch(dDio["In1_bPrdSta1"]==false,2)
        logMsg("In1_bPrdSta1触发:工位1信号被触发")
        //      x_bCanProuct[1]=true
        x_nWorkPlace=1
        return
      endIf
    endIf
  endIf

  //第二工位
  if dDio["In1_bPrdSta2"]==true
    delay(0.2)
    if watch(dDio["In1_bPrdSta2"]==true,0.1)
      if watch(dDio["In1_bPrdSta2"]==false,2)
        logMsg("In1_bPrdSta2触发:工位2信号被触发")
        //x_bCanProuct[2]=true
        x_nWorkPlace=2
        return
      endIf
    endIf
  endIf


  //第三工位
  if dDio["In2_bPrdSta3"]==true
    delay(0.2)
    if watch(dDio["In2_bPrdSta3"]==true,0.1)
      if watch(dDio["In2_bPrdSta3"]==false,2)
        logMsg("In2_bPrdSta3触发:工位3信号被触发")
        //      x_bCanProuct[3]=true
        x_nWorkPlace=3
        return
      endIf
    endIf
  endIf

  //第四工位
  if dDio["In2_bPrdSta4"]==true
    delay(0.2)
    if watch(dDio["In2_bPrdSta4"]==true,0.1)
      //      x_bCanProuct[4]=true
      if watch(dDio["In2_bPrdSta4"]==false,2)
        logMsg("In2_bPrdSta4触发:工位4信号被触发")
        x_nWorkPlace=4
        return
      endIf
    endIf
  endIf



end

--- ChoosehansPro.pgx ---
public program ChoosehansPro(num& x_nWorkPlace (dimensions=1), num& x_nProductIndex (dimensions=1), num& x_nMax[] (dimensions=1))
  local num l_nNum
begin
  //  //2013.10.30
  //  //通过数字量来选择产品
  //  //主要用来检测按钮触发
  //  //同工位多产品函数

  //2014.05.30





  //  x_nProductIndex=0
  //  x_nProductIndex=0
  //  l_nNum=0

  if x_nProductIndex>=x_nMax[x_nWorkPlace]
    x_nProductIndex=0
  endIf

  if x_nProductIndex>0
    x_nProductIndex=x_nProductIndex+1
    return

  endIf

  while true
    //工位1
    if dDio["In1_bPrdSta1"]==true and dDio["UsIn_bNull1"]==true and dDio["UsIn_bNull2"]==true
      delay(0.1)
      if dDio["In1_bPrdSta1"]==true and dDio["UsIn_bNull1"]==true and dDio["UsIn_bNull2"]==true
        //
        x_nProductIndex=1
        x_nWorkPlace=1
        return
      endIf
    endIf


    //工位2
    if dDio["In1_bPrdSta2"]==true and dDio["UsIn_bNull3"]==true and dDio["UsIn_bNull3"]==true
      delay(0.1)
      if dDio["In1_bPrdSta2"]==true and dDio["UsIn_bNull3"]==true and dDio["UsIn_bNull4"]==true
        //
        x_nProductIndex=1
        x_nWorkPlace=2
        return
      endIf
    endIf


    //工位3
    if dDio["In1_bPrdSta2"]==true and dDio["UsIn_bNull5"]==true and dDio["UsIn_bNull6"]==true
      delay(0.1)
      if dDio["In1_bPrdSta2"]==true and dDio["UsIn_bNull5"]==true and dDio["UsIn_bNull6"]==true
        //
        x_nProductIndex=1
        x_nWorkPlace=3
        return
      endIf
    endIf







    //2014.06.03
    //*************************************************************************
    //*************************************************************************

    //为大族定制
    //A1,A2,A3,A4
    if dDio["In1_bPrdSta1"]==true and dDio["UsIn_bNull1"]==true and dDio["UsIn_bNull2"]==true
      delay(0.1)
      if dDio["In1_bPrdSta1"]==true and dDio["UsIn_bNull1"]==true and dDio["UsIn_bNull2"]==true
        //
        x_nProductIndex=1
        x_nWorkPlace=1
        x_nMax[1]=4
        return
      endIf
    endIf


    //A1,A2
    if dDio["In1_bPrdSta1"]==true and dDio["UsIn_bNull1"]==true and dDio["UsIn_bNull2"]==true
      delay(0.1)
      if dDio["In1_bPrdSta1"]==true and dDio["UsIn_bNull1"]==true and dDio["UsIn_bNull2"]==true
        //
        x_nProductIndex=1
        x_nWorkPlace=1
        x_nMax[1]=2
        return
      endIf
    endIf

    //A3,A4
    if dDio["In1_bPrdSta1"]==true and dDio["UsIn_bNull1"]==true and dDio["UsIn_bNull2"]==true
      delay(0.1)
      if dDio["In1_bPrdSta1"]==true and dDio["UsIn_bNull1"]==true and dDio["UsIn_bNull2"]==true
        //
        x_nProductIndex=3
        x_nWorkPlace=1
        x_nMax[1]=4
        return
      endIf
    endIf

    //***********************************************************************************
    //**********************************************************************************



    delay(0)
  endWhile




end

--- ChooseMultPro.pgx ---
public program ChooseMultPro(num& x_nWorkPlace (dimensions=1), num& x_nProductIndex (dimensions=1))
  local num l_nNum
begin
  //2013.10.30
  //通过数字量来选择产品
  //主要用来检测按钮触发
  //同工位多产品函数
  //专为法利莱编写
  //需要外部PLC支持
  //DataBase中的变量需改变


  x_nProductIndex=0
  x_nProductIndex=0
  l_nNum=0


  wait(dDio["UsIn_bNull1"]==true or dDio["UsIn_bNull2"]==true or dDio["UsIn_bNull3"]==true or dDio["UsIn_bNull4"]==true or dDio["UsIn_bNull5"]==true or dDio["UsIn_bNull6"]==true or dDio["UsIn_bNull7"]==true or dDio["UsIn_bNull8"]==true)
  delay(0.2)
  //1，2，3，4对应工位1可能有的15种组合
  if dDio["UsIn_bNull1"]==true or dDio["UsIn_bNull2"]==true or dDio["UsIn_bNull3"]==true or dDio["UsIn_bNull4"]==true
    x_nWorkPlace=1
    l_nNum=sel(dDio["UsIn_bNull1"]==true,1,0)*1+l_nNum
    l_nNum=sel(dDio["UsIn_bNull2"]==true,1,0)*2+l_nNum
    l_nNum=sel(dDio["UsIn_bNull3"]==true,1,0)*4+l_nNum
    l_nNum=sel(dDio["UsIn_bNull4"]==true,1,0)*8+l_nNum
  endIf
  //5，6，7，8对应工位2可能有的15种组合
  if dDio["UsIn_bNull5"]==true or dDio["UsIn_bNull6"]==true or dDio["UsIn_bNull7"]==true or dDio["UsIn_bNull8"]==true
    x_nWorkPlace=2
    l_nNum=sel(dDio["UsIn_bNull5"]==true,1,0)*1+l_nNum
    l_nNum=sel(dDio["UsIn_bNull6"]==true,1,0)*2+l_nNum
    l_nNum=sel(dDio["UsIn_bNull7"]==true,1,0)*4+l_nNum
    l_nNum=sel(dDio["UsIn_bNull8"]==true,1,0)*8+l_nNum
  endIf

  if l_nNum>15
    x_nWorkPlace=-1
    return
  endIf

  x_nProductIndex=l_nNum
  logMsg("工位"+toString("",x_nWorkPlace)+":"+"选择产品号"+toString("",x_nProductIndex))

  dDio["UsO_bNull1"]=true
  wait(dDio["UsIn_bNull1"]==false and dDio["UsIn_bNull2"]==false and dDio["UsIn_bNull3"]==false and dDio["UsIn_bNull4"]==false and dDio["UsIn_bNull5"]==false and dDio["UsIn_bNull6"]==false and dDio["UsIn_bNull7"]==false and dDio["UsIn_bNull8"]==false)
  dDio["UsO_bNull1"]=false

  logMsg("工位选择产品完成")

end

--- CloseWeld.pgx ---
public program CloseWeld(num x_nWeldTime)
begin
  //收弧关闭



  //  x_nWeldTime=max(0,min(0.999,x_nWeldTime))
  //
  //  //动作
  //  if !x_bAction
  //   // $waitEndMove(x_nWeldTime)
  //
  ////    dDio["UsO_bNull5"]=true
  ////    call Digtal2AnalogS(0)
  //
  //  endIf

  //2015.09.08
  //为收弧修改时间
  // waitEndMove()

  if dDio["UsO_bNull5"]==false and dDio["UsO_bNull4"]==true

    dDio["UsO_bNull5"]=true
    // delay(0.1)
    //用户自定义IO强制设为0
    call Digtal2AnalogS(0)
    delay(0.05)
  endIf

  //用户自定义IO强制设为0
  dDio["UsO_bNull5"]=false
  //  delay(0.1)
  call Digtal2AnalogS(0)
  //delay(0.)


end

--- Digtal2Analog.pgx ---
public program Digtal2Analog()
  local num l_nIndexX
  local num l_nIndexY
  local num l_nNum
  local string l_sIOName
begin

  //数字量转换为模拟量

  //  for l_nIndexY=0 to 4
  //    l_nNum=0
  //    for l_nIndexX =0 to 15
  //      call IOName(67+l_nIndexX+l_nIndexY*16,l_sIOName)
  //      if (67+l_nIndexX+l_nIndexY*16)<135
  //        l_nNum=l_nNum+sel(dDio[l_sIOName]==true,1,0)*power(2,l_nIndexX)
  //      endIf
  //    endFor
  //    call IOName(159+l_nIndexY,l_sIOName)
  //    aioSet(aAio[l_sIOName],l_nNum)
  //  //  delay(0)
  //  endFor
  //


  call Digtal2AnalogS(0)
  call Digtal2AnalogS(1)
  call Digtal2AnalogS(2)
  call Digtal2AnalogS(3)
  call Digtal2AnalogS(4)

end

--- Digtal2AnalogS.pgx ---
public program Digtal2AnalogS(num x_nId (dimensions=1))
  local num l_nIndexX
  local num l_nIndexY
  local num l_nNum
  local string l_sIOName
begin

  //数字量转换为模拟量

  //0 67到82
  //1 83到98
  //2 99到114
  //3 115到130
  //4 131到146


  x_nId=min(4,max(0,x_nId))
  for l_nIndexY=x_nId to x_nId
    l_nNum=0
    for l_nIndexX=0 to 15
      call IOName(67+l_nIndexX+l_nIndexY*16,l_sIOName)
      if (67+l_nIndexX+l_nIndexY*16)<135
        l_nNum=l_nNum+sel(dDio[l_sIOName]==true,1,0)*power(2,l_nIndexX)
      endIf
    endFor
    call IOName(159+l_nIndexY,l_sIOName)
    aioSet(aAio[l_sIOName],l_nNum)
    delay(0)
  endFor



























end

--- ExtraContrAxis.pgx ---
public program ExtraContrAxis(num x_nPosition, bool& x_bRes)
begin

  //2014.11.25
  //利用外部PLC来控制异步外部第七轴的运动
  //客户可以重构此函数
  //只支持四个位置，1，2，3，4
  //使用说明请查看 lasman使用手册 PLC控制外部轴
  //每条路径对应不同的外部轴位置


  x_bRes=false

  //检查参数是否合法
  if roundDown(x_nPosition)!=x_nPosition or x_nPosition<0 or x_nPosition>4
    return
  endIf



  //等待手臂到位信号
  wait(dDio["UsIn_bNull1"]==true)


  //让机械手臂停止
  if x_nPosition!=0
    waitEndMove()
  else
    x_bRes=true
    return
  endIf

  switch x_nPosition

    //转盘第一位置
    case 1
      dDio["UsO_bNull3"]=true
      delay(0.5)
      dDio["UsO_bNull3"]=false
    break


    //转盘第二位置
    case 2
      dDio["UsO_bNull4"]=true
      delay(0.5)
      dDio["UsO_bNull4"]=false

    break

    //转盘第二位置
    case 3
      dDio["UsO_bNull5"]=true
      delay(0.5)
      dDio["UsO_bNull5"]=false
    break

    //转盘第三位置
    case 4
      dDio["UsO_bNull6"]=true
      delay(0.5)
      dDio["UsO_bNull6"]=false
    break



  endSwitch



  if x_nPosition!=0
    delay(0.5)
    //位置确认信号
    dDio["UsO_bNull1"]=true
    delay(0.5)
    dDio["UsO_bNull1"]=false
    delay(0.5)
    //位置启动
    dDio["UsO_bNull7"]=true
    delay(0.5)
    dDio["UsO_bNull7"]=false
    delay(0.5)
  endIf


  //等待到位信号
  wait(dDio["UsIn_bNull1"]==true)

  x_bRes=true
end

--- GasChoose.pgx ---
public program GasChoose(num x_nGasIndex)
begin
  //2015.05.28
  //气体选择，为特定的气体做选择


  if roundDown(x_nGasIndex)!=roundUp(x_nGasIndex)
      x_nGasIndex=0
  endIf


  switch  x_nGasIndex
    case 0
      dDio["UsO_bNull5"]=false
      dDio["UsO_bNull6"]=false
      dDio["UsO_bNull8"]=false

    break

    case 1
      dDio["UsO_bNull5"]=true
      dDio["UsO_bNull6"]=false
      dDio["UsO_bNull8"]=false
    break


    case 2
      dDio["UsO_bNull5"]=false
      dDio["UsO_bNull6"]=true
      dDio["UsO_bNull8"]=false
    break


    case 3
      dDio["UsO_bNull5"]=false
      dDio["UsO_bNull6"]=false
      dDio["UsO_bNull8"]=true

    break





  endSwitch

  call Digtal2Analog()






end

--- GetAxis7Pos.pgx ---
public program GetAxis7Pos(num& x_nPosition (dimensions=1), num x_nPrecent (dimensions=1))
begin

  dDio["O4_b7RecordPos"]=true
  delay(0.05)
  dDio["O4_b7RecordPos"]=false

  x_nPosition=aioGet(aAio["In4_a7CurPosH"])*power(2,16)+aioGet(aAio["In4_a7CurPosL"])
  x_nPosition=x_nPosition/max(x_nPrecent,0.001)

end

--- GetAxis8Pos.pgx ---
public program GetAxis8Pos(num& x_nPosition (dimensions=1), num x_nPrecent (dimensions=1))
begin

  dDio["O4_b8RecordPos"]=true
  delay(0.05)
  dDio["O4_b8RecordPos"]=false


  x_nPosition=aioGet(aAio["In4_a8CurPosH"])*power(2,16)+aioGet(aAio["In4_a8CurPosL"])
  x_nPosition=x_nPosition/max(x_nPrecent,0.001)

end

--- GetAxisStatus.pgx ---
public program GetAxisStatus(bool& x_bBPower (dimensions=1), bool& x_nAlarm (dimensions=1), bool& x_nBackHome (dimensions=1))
begin
  x_bBPower=(dDio["In4_b7MotorPower"]==true)
  x_nAlarm=(dDio["In4_b7MotorError"]==true)
  x_nBackHome=(dDio["In4_b7BackHome"]==true)
end

--- GetKeyIO.pgx ---
public program GetKeyIO(bool& x_AirOn (dimensions=1), bool& x_bFollowOn (dimensions=1), bool& x_bLaserOn (dimensions=1))
  local string l_sS
begin

  //气体
  call IOName(70,l_sS)
  x_AirOn=dDio[l_sS]==true


  //随动
  call IOName(68,l_sS)
  x_bFollowOn=dDio[l_sS]==true


  //焊接
  if bWeldEnable
    call IOName(79,l_sS)
    x_bLaserOn=dDio[l_sS]==true

  else
    //   切割
    call IOName(67,l_sS)
    x_bLaserOn=dDio[l_sS]==true
  endIf

end

--- GetPreset.pgx ---
public program GetPreset(num& x_nPreset[] (dimensions=1), num x_nPrecent (dimensions=1), num x_nPWMH (dimensions=1), num x_nPWML (dimensions=1))
  local num l_nNum
  local num l_nPWM
begin

  x_nPreset[0]=aioGet(aAio["O1_aLasPwr"])
  x_nPreset[1]=aioGet(aAio["O1_aFPWM"])
  x_nPreset[2]=aioGet(aAio["O1_aPMW"])
  x_nPreset[3]=aioGet(aAio["O1_aAirPress"])
  x_nPreset[4]=aioGet(aAio["O2_aFollowSensitive"])

  for l_nNum=0 to 4
    if l_nNum==1
      //强制设置为1500
      l_nPWM=x_nPWMH-x_nPWML
      l_nPWM=sel(l_nPWM<1,1,l_nPWM)
      x_nPreset[1]=(x_nPreset[1]-x_nPWML)/l_nPWM*100
    else
      if l_nNum!=2
        x_nPreset[l_nNum]=round(x_nPreset[l_nNum]/max(x_nPrecent,1)*100)
      endIf
    endIf
  endFor



end

--- Init.pgx ---
public program Init()
  local num l_nNum
begin
  //LasMAN modbus表格的初始化




  //dDio["In1_bPowerOn"]=false
  //dDio["In1_bStartCycl"]=false
  //dDio["In1_bStopCycl"]=false
  //dDio["In1_bHome"]=false
  //dDio["In1_bEndCycl"]=false
  //dDio["In1_bPrdSta1"]=false
  //dDio["In1_bPrdSta2"]=false
  //dDio["In1_bPausCycl"]=false
  //dDio["In1_bOutAlarm"]=false
  //dDio["In1_bReset"]=false
  //dDio["In1_bPeripheralReady"]=false
  //dDio["In1_bNull1"]=false
  //dDio["In1_bNull2"]=false
  //dDio["In1_bNull3"]=false
  //dDio["UsIn_bNull1"]=false
  //dDio["UsIn_bNull2"]=false
  //dDio["UsIn_bNull3"]=false
  //dDio["UsIn_bNull4"]=false
  //dDio["UsIn_bNull5"]=false
  //dDio["UsIn_bNull6"]=false
  //dDio["UsIn_bNull7"]=false
  //dDio["UsIn_bNull8"]=false
  //dDio["In2_bPrdSta3"]=false
  //dDio["In2_bPrdSta4"]=false
  //dDio["In2_bAirAlarm"]=false
  //dDio["In2_bCollisonAlarm"]=false
  //dDio["In2_bLaserAlarm"]=false
  //dDio["In2_bContactAlarm"]=false
  //dDio["In2_bRasterOn"]=false
  //dDio["In2_bNull1"]=false
  //dDio["In2_bNull2"]=false
  //dDio["In2_bNull3"]=false
  //dDio["In2_bNull4"]=false
  //dDio["In2_bNull5"]=false
  //dDio["In2_bNull6"]=false
  //dDio["In2_bNull7"]=false
  //dDio["In2_bNull8"]=false
  //dDio["In2_bNull9"]=false
  //dDio["In7_bUpLimit_7"]=false
  //dDio["In7_bDownLimit_7"]=false
  //dDio["In7_bHomeLimit_7"]=false
  //dDio["In7_bNull1"]=false
  //dDio["In8_bUpLimit_8"]=false
  //dDio["In8_bDownLimit_8"]=false
  //dDio["In8_bHomeLimit_8"]=false
  //dDio["In8_bNull1"]=false
  //dDio["In4_b7Reached"]=false
  //dDio["In4_b7BackHome"]=false
  //dDio["In4_b7HomeDone"]=false
  //dDio["In4_b7MotorPower"]=false
  //dDio["In4_b7IsHome"]=false
  //dDio["In4_b7MotorError"]=false
  //dDio["In4_b8Reached"]=false
  //dDio["In4_b8BackHome"]=false
  //dDio["In4_b8HomeDone"]=false
  //dDio["In4_b8MotorPower"]=false
  //dDio["In4_b8IsHome"]=false
  //dDio["In4_b8MotorError"]=false
  //dDio["In4_bNull1"]=false
  //dDio["In4_bNull2"]=false
  //dDio["In4_bNull3"]=false
  //dDio["In4_bNull4"]=false
  //dDio["In4_bNull5"]=false
  //dDio["In4_bNull6"]=false
  //dDio["In4_bNull7"]=false
  //dDio["In4_bNull8"]=false

  //所有数字量输出为false
  dDio["O1_bLaserOn"]=false
  dDio["O1_bFollowOn"]=false
  dDio["O1_bFollowDone"]=false
  dDio["O1_bAirOn"]=false
  dDio["O1_bNull1"]=false
  dDio["O1_bRedLamp"]=false
  dDio["O1_bYellowLamp"]=false
  dDio["O1_bGreenLamp"]=false
  dDio["O1_bAlarm"]=false
  dDio["UsO_bNull1"]=false
  dDio["UsO_bNull2"]=false
  dDio["UsO_bNull3"]=false
  dDio["UsO_bNull4"]=false
  dDio["UsO_bNull5"]=false
  dDio["UsO_bNull6"]=false
  dDio["UsO_bNull7"]=false
  dDio["UsO_bNull8"]=false
  dDio["O2_bSta1Stat"]=false
  dDio["O2_bSta2Stat"]=false
  dDio["O2_bSta3Stat"]=false
  dDio["O2_bSta4Stat"]=false
  dDio["O2_bProCode1"]=false
  dDio["O2_bProCode2"]=false
  dDio["O2_bProCode3"]=false
  dDio["O2_bFollowHeigh1"]=false
  dDio["O2_bFollowHeigh2"]=false
  dDio["O2_bFollowHeigh3"]=false
  dDio["O2_bAxisPos1"]=false
  dDio["O2_bAxisPos2"]=false
  dDio["O2_bAxisPos3"]=false
  dDio["O2_bNull1"]=false
  dDio["O2_bNull2"]=false
  dDio["O2_bNull3"]=false
  dDio["O7_bAxis7Pulse"]=false
  dDio["O7_bAxis7Direction"]=false
  dDio["O7_bNull1"]=false
  dDio["O7_bNull2"]=false
  dDio["O7_bNull3"]=false
  dDio["O8_bAxis8Pulse"]=false
  dDio["O8_bAxis8Direction"]=false
  dDio["O8_bNull1"]=false
  dDio["O8_bNull2"]=false
  dDio["O8_bNull3"]=false
  dDio["O4_b7RecordPos"]=false
  dDio["O4_b7MoveToPos"]=false
  dDio["O4_b7ResetError"]=false
  dDio["O4_b7ChkHome"]=false
  dDio["O4_b7AxisHome"]=false
  dDio["O4_b7MoveDir"]=false
  dDio["O4_b7MoveDirM"]=false
  dDio["O4_b7StopMotor"]=false
  dDio["O4_bHome"]=false
  dDio["O4_b8RecordPos"]=false
  dDio["O4_b8MoveToPos"]=false
  dDio["O4_b8ResetError"]=false
  dDio["O4_b8ChkHome"]=false
  dDio["O4_b8AxisHome"]=false
  dDio["O4_b8MoveDir"]=false
  dDio["O4_b8MoveDirM"]=false
  dDio["O4_b8StopMotor"]=false
  dDio["O4_bNull1"]=false
  dDio["O4_bNull2"]=false
  dDio["O4_bNull3"]=false
  dDio["O4_bNull4"]=false
  dDio["O4_bNull5"]=false
  dDio["O4_bNull6"]=false
  dDio["O4_bNull7"]=false
  dDio["O4_bNull8"]=false





  //所有模拟量输出为0
  aioSet(aAio["O1_aLasPwr"],0)
  aioSet(aAio["O1_aAirPress"],0)
  aioSet(aAio["O1_aFPWM"],0)
  aioSet(aAio["O1_aPMW"],0)
  aioSet(aAio["O2_aFollowSensitive"],0)
  aioSet(aAio["O2_aNull"],0)
  //aioSet(aAio["In4_a7CurPosL"] ,0)
  //aioSet(aAio["In4_a7CurPosH"] ,0)
  //aioSet(aAio["In4_a8CurPosL"] ,0)
  //aioSet(aAio["In4_a8CurPosH"] ,0)
  aioSet(aAio["O4_a7Velocity"],0)
  aioSet(aAio["O4_a7JogVelo"],0)
  aioSet(aAio["O4_a7MoveDis"],0)
  aioSet(aAio["O4_a7AiHomeH"],0)
  aioSet(aAio["O4_a7AiHomeL"],0)
  aioSet(aAio["O4_a7MovePosL"],0)
  aioSet(aAio["O4_a7MovePosH"],0)
  aioSet(aAio["O4_a8Velocity"],0)
  aioSet(aAio["O4_a8JogVelo"],0)
  aioSet(aAio["O4_a8MoveDis"],0)
  aioSet(aAio["O4_a8AiHomeH"],0)
  aioSet(aAio["O4_a8AiHomeL"],0)
  aioSet(aAio["O4_a8MovePosL"],0)
  aioSet(aAio["O4_a8MovePosH"],0)
  aioSet(aAio["Out_a66_81"],0)
  aioSet(aAio["Out_a82_97"],0)
  aioSet(aAio["Out_a98_113"],0)
  aioSet(aAio["Out_a114_129"],0)
  aioSet(aAio["Out_a130_133"],0)
  //aioSet(aAio["In_aVersion"] ,0)

  resize(sIOName,1,167)
  for l_nNum=0 to 166
    call IOName(l_nNum,sIOName[l_nNum])
  endFor

  resize(bDigtal,1,167)
  for l_nNum=0 to 166
    call IsDigtal(l_nNum,bDigtal[l_nNum])
  endFor


end

--- IOName.pgx ---
public program IOName(num x_nId (dimensions=1), string& x_sName (dimensions=1))
begin

  x_sName=""
  switch x_nId
    //×××××××××××××××××××××××××××××××××××××××××××××
    //输入
    case 0
      x_sName="无"
    break
    case 1
      x_sName="In1_bPowerOn"
    break
    case 2
      x_sName="In1_bStartCycl"
    break
    case 3
      x_sName="In1_bStopCycl"
    break
    case 4
      x_sName="In1_bHome"
    break
    case 5
      x_sName="In1_bEndCycl"
    break
    case 6
      x_sName="In1_bPrdSta1"
    break
    case 7
      x_sName="In1_bPrdSta2"
    break
    case 8
      x_sName="In1_bPausCycl"
    break
    case 9
      x_sName="In1_bOutAlarm"
    break
    case 10
      x_sName="In1_bReset"
    break
    case 11
      x_sName="In1_bPeripheralReady"
    break
    case 12
      x_sName="In1_bNull1"
    break
    case 13
      x_sName="In1_bNull2"
    break
    case 14
      x_sName="In1_bNull3"
    break
    case 15
      x_sName="UsIn_bNull1"
    break
    case 16
      x_sName="UsIn_bNull2"
    break
    case 17
      x_sName="UsIn_bNull3"
    break
    case 18
      x_sName="UsIn_bNull4"
    break
    case 19
      x_sName="UsIn_bNull5"
    break
    case 20
      x_sName="UsIn_bNull6"
    break
    case 21
      x_sName="UsIn_bNull7"
    break
    case 22
      x_sName="UsIn_bNull8"
    break
    case 23
      x_sName="In2_bPrdSta3"
    break
    case 24
      x_sName="In2_bPrdSta4"
    break
    case 25
      x_sName="In2_bAirAlarm"
    break
    case 26
      x_sName="In2_bCollisonAlarm"
    break
    case 27
      x_sName="In2_bLaserAlarm"
    break
    case 28
      x_sName="In2_bContactAlarm"
    break
    case 29
      x_sName="In2_bRasterOn"
    break
    case 30
      x_sName="In2_bNull1"
    break
    case 31
      x_sName="In2_bNull2"
    break
    case 32
      x_sName="In2_bNull3"
    break
    case 33
      x_sName="In2_bNull4"
    break
    case 34
      x_sName="In2_bNull5"
    break
    case 35
      x_sName="In2_bNull6"
    break
    case 36
      x_sName="In2_bNull7"
    break
    case 37
      x_sName="In2_bNull8"
    break
    case 38
      x_sName="In2_bNull9"
    break
    case 39
      x_sName="In7_bUpLimit_7"
    break
    case 40
      x_sName="In7_bDownLimit_7"
    break
    case 41
      x_sName="In7_bHomeLimit_7"
    break
    case 42
      x_sName="In7_bNull1"
    break
    case 43
      x_sName="In8_bUpLimit_8"
    break
    case 44
      x_sName="In8_bDownLimit_8"
    break
    case 45
      x_sName="In8_bHomeLimit_8"
    break
    case 46
      x_sName="In8_bNull1"
    break
    case 47
      x_sName="In4_b7Reached"
    break
    case 48
      x_sName="In4_b7BackHome"
    break
    case 49
      x_sName="In4_b7HomeDone"
    break
    case 50
      x_sName="In4_b7MotorPower"
    break
    case 51
      x_sName="In4_b7IsHome"
    break
    case 52
      x_sName="In4_b7MotorError"
    break
    case 53
      x_sName="In4_b8Reached"
    break
    case 54
      x_sName="In4_b8BackHome"
    break
    case 55
      x_sName="In4_b8HomeDone"
    break
    case 56
      x_sName="In4_b8MotorPower"
    break
    case 57
      x_sName="In4_b8IsHome"
    break
    case 58
      x_sName="In4_b8MotorError"
    break
    case 59
      x_sName="In4_bNull1"
    break
    case 60
      x_sName="In4_bNull2"
    break
    case 61
      x_sName="In4_bNull3"
    break
    case 62
      x_sName="In4_bNull4"
    break
    case 63
      x_sName="In4_bNull5"
    break
    case 64
      x_sName="In4_bNull6"
    break
    case 65
      x_sName="In4_bNull7"
    break
    case 66
      x_sName="In4_bNull8"
    break
    //×××××××××××××××××××××××××××××××××××××××××××××××××××
    //0输出
    case 67
      x_sName="O1_bLaserOn"
    break
    case 68
      x_sName="O1_bFollowOn"
    break
    case 69
      x_sName="O1_bFollowDone"
    break
    case 70
      x_sName="O1_bAirOn"
    break
    case 71
      x_sName="O1_bNull1"
    break
    case 72
      x_sName="O1_bRedLamp"
    break
    case 73
      x_sName="O1_bYellowLamp"
    break
    case 74
      x_sName="O1_bGreenLamp"
    break
    case 75
      x_sName="O1_bAlarm"
    break
    case 76
      x_sName="UsO_bNull1"
    break
    case 77
      x_sName="UsO_bNull2"
    break
    case 78
      x_sName="UsO_bNull3"
    break
    case 79
      x_sName="UsO_bNull4"
    break
    case 80
      x_sName="UsO_bNull5"
    break
    case 81
      x_sName="UsO_bNull6"
    break
    case 82
      x_sName="UsO_bNull7"
    break


    //1输出
    case 83
      x_sName="UsO_bNull8"
    break

    case 84
      x_sName="O2_bSta1Stat"
    break
    case 85
      x_sName="O2_bSta2Stat"
    break
    case 86
      x_sName="O2_bSta3Stat"
    break
    case 87
      x_sName="O2_bSta4Stat"
    break
    case 88
      x_sName="O2_bProCode1"
    break
    case 89
      x_sName="O2_bProCode2"
    break
    case 90
      x_sName="O2_bProCode3"
    break
    case 91
      x_sName="O2_bFollowHeigh1"
    break
    case 92
      x_sName="O2_bFollowHeigh2"
    break
    case 93
      x_sName="O2_bFollowHeigh3"
    break
    case 94
      x_sName="O2_bAxisPos1"
    break
    case 95
      x_sName="O2_bAxisPos2"
    break
    case 96
      x_sName="O2_bAxisPos3"
    break
    case 97
      x_sName="O2_bNull1"
    break
    case 98
      x_sName="O2_bNull2"
    break

    //3输出
    case 99
      x_sName="O2_bNull3"
    break
    case 100
      x_sName="O7_bAxis7Pulse"
    break
    case 101
      x_sName="O7_bAxis7Direction"
    break
    case 102
      x_sName="O7_bNull1"
    break
    case 103
      x_sName="O7_bNull2"
    break
    case 104
      x_sName="O7_bNull3"
    break
    case 105
      x_sName="O8_bAxis8Pulse"
    break
    case 106
      x_sName="O8_bAxis8Direction"
    break
    case 107
      x_sName="O8_bNull1"
    break
    case 108
      x_sName="O8_bNull2"
    break
    case 109
      x_sName="O8_bNull3"
    break
    case 110
      x_sName="O4_b7RecordPos"
    break
    case 111
      x_sName="O4_b7MoveToPos"
    break
    case 112
      x_sName="O4_b7ResetError"
    break
    case 113
      x_sName="O4_b7ChkHome"
    break
    case 114
      x_sName="O4_b7AxisHome"
    break

    //4 Digtal2Analog
    case 115
      x_sName="O4_b7MoveDir"
    break
    case 116
      x_sName="O4_b7MoveDirM"
    break
    case 117
      x_sName="O4_b7StopMotor"
    break
    case 118
      x_sName="O4_bHome"
    break
    case 119
      x_sName="O4_b8RecordPos"
    break
    case 120
      x_sName="O4_b8MoveToPos"
    break
    case 121
      x_sName="O4_b8ResetError"
    break
    case 122
      x_sName="O4_b8ChkHome"
    break
    case 123
      x_sName="O4_b8AxisHome"
    break
    case 124
      x_sName="O4_b8MoveDir"
    break
    case 125
      x_sName="O4_b8MoveDirM"
    break
    case 126
      x_sName="O4_b8StopMotor"
    break
    case 127
      x_sName="O4_bNull1"
    break
    case 128
      x_sName="O4_bNull2"
    break
    case 129
      x_sName="O4_bNull3"
    break
    case 130
      x_sName="O4_bNull4"
    break
    case 131
      x_sName="O4_bNull5"
    break
    case 132
      x_sName="O4_bNull6"
    break
    case 133
      x_sName="O4_bNull7"
    break
    case 134
      x_sName="O4_bNull8"
    break

    //模拟量
    case 135
      x_sName="O1_aLasPwr"
    break
    case 136
      x_sName="O1_aAirPress"
    break
    case 137
      x_sName="O1_aFPWM"
    break
    case 138
      x_sName="O1_aPMW"
    break
    case 139
      x_sName="O2_aFollowSensitive"
    break
    case 140
      x_sName="O2_aNull"
    break
    case 141
      x_sName="In4_a7CurPosL"
    break
    case 142
      x_sName="In4_a7CurPosH"
    break
    case 143
      x_sName="In4_a8CurPosL"
    break
    case 144
      x_sName="In4_a8CurPosH"
    break
    case 145
      x_sName="O4_a7Velocity"
    break
    case 146
      x_sName="O4_a7JogVelo"
    break
    case 147
      x_sName="O4_a7MoveDis"
    break
    case 148
      x_sName="O4_a7AiHomeH"
    break
    case 149
      x_sName="O4_a7AiHomeL"
    break
    case 150
      x_sName="O4_a7MovePosL"
    break
    case 151
      x_sName="O4_a7MovePosH"
    break
    case 152
      x_sName="O4_a8Velocity"
    break
    case 153
      x_sName="O4_a8JogVelo"
    break
    case 154
      x_sName="O4_a8MoveDis"
    break
    case 155
      x_sName="O4_a8AiHomeH"
    break
    case 156
      x_sName="O4_a8AiHomeL"
    break
    case 157
      x_sName="O4_a8MovePosL"
    break
    case 158
      x_sName="O4_a8MovePosH"
    break
    case 159
      x_sName="Out_a66_81"
    break
    case 160
      x_sName="Out_a82_97"
    break
    case 161
      x_sName="Out_a98_113"
    break
    case 162
      x_sName="Out_a114_129"
    break
    case 163
      x_sName="Out_a130_133"
    break
    case 164
      x_sName="In_aVersion"
    break



    //额外添加
    case 165
      x_sName="延时"
    break

    //收弧时间
    case 166
      x_sName="收弧时间"
    break

    //收弧长度
    case 167
      x_sName="收弧长度"
    break



  endSwitch

end

--- IOvalue.pgx ---
program IOvalue(num x_nIOid (dimensions=1), num x_nIoValue (dimensions=1))
  local bool l_IsInput
  local bool l_bFollowOn
  local bool l_bGasOn
  local bool l_bLaserOn
  local string l_sName
begin
  //2014.05.23
  //通过对输入信号进行处理
  //



  //0 表示无

  //165表示 延时

  x_nIoValue=max(x_nIoValue,0)


  //无动作
  if x_nIOid<=0 or x_nIOid>168
    return
  endIf

  //延时
  if x_nIOid==165
    waitEndMove()
    delay(max(0,x_nIoValue))
    return
  endIf


  //焊接收弧时间
  if x_nIOid==166
    //    delay(max(0,x_nIoValue))
    // $waitEndMove(max(0,min(0.999,x_nIoValue))*-1)
    //$waitEndMove(-2)
    return
  endIf


  //焊接收弧长度
  if x_nIOid==167
    //    delay(max(0,x_nIoValue))
    // $waitEndMove(max(0,min(0.999,x_nIoValue))*-1)
    //$waitEndMove(-2)
    return
  endIf



  x_nIoValue=round(x_nIoValue)
  call IsInput(x_nIOid,l_IsInput)
  call IOName(x_nIOid,l_sName)
  if l_IsInput
    //*********************************************************
    //2014.05.23
    //对于输入信号进行判断
    while !isEmpty()
      if find(l_sName,"_b")>=0
        if dDio[l_sName]==(x_nIoValue>=1)
          return
        endIf

        //  wait(dDio[l_sName]==(x_nIoValue>=1) or !isEmpty())
      else
        if aioGet(aAio[l_sName])==x_nIoValue
          return
        endIf
      endIf
      delay(0)
    endWhile

    call GetKeyIO(l_bGasOn,l_bFollowOn,l_bLaserOn)


    //如果有等待信号，那么激光则关
    if !bWaitActionOff
      call KeyDigtalIO(l_bGasOn,l_bFollowOn,false,0,0)
    endIf
    if find(l_sName,"_b")>=0
      wait(dDio[l_sName]==(x_nIoValue>=1))
    else
      wait(aioGet(aAio[l_sName])==x_nIoValue)
    endIf
    call KeyDigtalIO(l_bGasOn,l_bFollowOn,l_bLaserOn,0,0)
    //**************************
    //******************************************************************
  else
    if find(l_sName,"_b")>=0
      dDio[l_sName]=(x_nIoValue>=1)
    else
      aioSet(aAio[l_sName],x_nIoValue)
    endIf

  endIf


end

--- IsDigtal.pgx ---
program IsDigtal(num x_nIOid (dimensions=1), bool& x_bRes (dimensions=1))
begin
  x_bRes=x_nIOid<=134

end

--- IsInput.pgx ---
program IsInput(num x_nIOid (dimensions=1), bool& x_bRes (dimensions=1))
begin

  x_bRes=false
  switch true

    //序号为0
    //    case x_nIOid==0
    //      x_bRes=true
    //    break

    //数字量输入
    case x_nIOid>0 and x_nIOid<67
      x_bRes=true
    break


    //数字量输出
    case x_nIOid>134 and x_nIOid<=140
      x_bRes=false
    break

    //数字量输入
    case x_nIOid>140 and x_nIOid<=144
      x_bRes=true
    break

    //数字量输出
    case x_nIOid>144 and x_nIOid<=164
      x_bRes=false
    break

    //延时等待
    case x_nIOid==165
      x_bRes=true
    break


    //收弧时间
    case x_nIOid==166
      x_bRes=true
    break


    //收弧长度
    case x_nIOid==167
      x_bRes=false
    break


    default
    break
  endSwitch

end

--- KeyDigtalIO.pgx ---
public program KeyDigtalIO(bool x_bGas, bool x_bFollow, bool x_bLaser, num x_nGasDelay, num x_nFollowDelay)
begin
  //激光，随动，气体的能使信号
  //在激光切割中进行了定制

  //×××××××××××××××××××××××××××××
  //客户可以定制开气开随动开激光

  //气体
  if dDio["O1_bAirOn"]!=x_bGas
    dDio["O1_bAirOn"]=x_bGas
    call Digtal2AnalogS(0)
    if x_bGas
      delay(min(max(x_nGasDelay,0),20))
      logMsg("O1_bAirOn触发,气体开")
    else
      logMsg("O1_bAirOn触发,气体关")
    endIf
  endIf



  //随动
  if dDio["O1_bFollowOn"]!=x_bFollow
    //*****************************
    //抬枪信号
    //2014.06.06
    if bGunUp
      dDio["UsO_bNull1"]=x_bFollow
      if x_bFollow
        delay(0.1)
      endIf
    endIf
    //*****************************
    dDio["O1_bFollowOn"]=x_bFollow
    call Digtal2AnalogS(0)
    if x_bFollow
      if bWaitFollowDown
          logMsg("等待In1_bPeripheralReady为true")
        wait(dDio["In1_bPeripheralReady"]==true)
      endIf
      delay(min(max(x_nFollowDelay,0),20))
      //等待随动到位信号
      logMsg("O1_bFollowOn触发,随动开")
    else
      logMsg("O1_bFollowOn触发,随动关")
    endIf
  endIf





  //切割激光开与关
  if dDio["O1_bLaserOn"]!=x_bLaser
    dDio["O1_bLaserOn"]=x_bLaser
    call Digtal2AnalogS(0)
    if x_bLaser
      logMsg("O1_bLaserOn触发,激光开")
    else
      logMsg("O1_bLaserOn触发,激光关")
    endIf
  endIf


  //焊接激光开与关
  if bWeldEnable
    if dDio["UsO_bNull4"]!=x_bLaser
      dDio["UsO_bNull4"]=x_bLaser
      call Digtal2AnalogS(0)
      if x_bLaser
        logMsg("UsO_bNull4触发,激光开")
      else
        logMsg("UsO_bNull4触发,激光关")
      endIf
    endIf

  endIf



end

--- Light.pgx ---
public program Light(num x_nType (dimensions=1))
  local string l_sS
begin
  //对指示灯进行设置

  //0 红灯亮
  //1黄灯亮
  //2 绿灯亮


  //红
  call IOName(72,l_sS)
  dDio[l_sS]=(x_nType==0)
  //黄
  call IOName(73,l_sS)
  dDio[l_sS]=(x_nType==1)
  //绿
  call IOName(74,l_sS)
  dDio[l_sS]=(x_nType==2)
  //报警
  call IOName(75,l_sS)
  dDio[l_sS]=(x_nType==0)


end

--- MatchSpdPreset.pgx ---
public program MatchSpdPreset(num& x_nPreset[] (dimensions=2), num x_nIndex (dimensions=1), num x_nPercent (dimensions=1), num x_nHZHight (dimensions=1), num x_nHZLow (dimensions=1))
  local num l_nNum
begin


  //激光工艺设置
  if x_nIndex>0 and x_nIndex<201
    x_nIndex=roundDown(x_nIndex)
    aioSet(aAio["O1_aLasPwr"],x_nPreset[x_nIndex,0]/100*x_nPercent)
    aioSet(aAio["O1_aAirPress"],x_nPreset[x_nIndex,1]/100*x_nPercent)
    //  aioSet(aAio["O1_aFPWM"],x_nPreset[x_nIndex,2]/100*x_nPercent)
    aioSet(aAio["O1_aFPWM"],x_nPreset[x_nIndex,2]*(x_nHZHight-x_nHZLow)/100+x_nHZLow)
    //  aioSet(aAio["O1_aPMW"],x_nPreset[x_nIndex,3]/100*x_nPercent)
    aioSet(aAio["O1_aPMW"],min(max(x_nPreset[x_nIndex,3],0),100))
    aioSet(aAio["O2_aFollowSensitive"],x_nPreset[x_nIndex,4]/100*x_nPercent)
    //  aioSet(aAio["O1_aLasPwr"],x_nPreset[x_nIndex,4])

    if !bDigFollowHight
      return
    endIf
    //2014.05.27
    //对随动高度进行转换
    //0 false false false
    //1~12  true false false
    //13~25  true false false
    //26~38  true false false


    // l_nNum=round(x_nPreset[x_nIndex,4]/12.5)
    l_nNum=round(x_nPreset[x_nIndex,4])
    switch l_nNum
      case 0
        dDio["O2_bFollowHeigh1"]=false
        dDio["O2_bFollowHeigh2"]=false
        dDio["O2_bFollowHeigh3"]=false
      break

      case 1
        dDio["O2_bFollowHeigh1"]=true
        dDio["O2_bFollowHeigh2"]=false
        dDio["O2_bFollowHeigh3"]=false
      break
      case 2
        dDio["O2_bFollowHeigh1"]=false
        dDio["O2_bFollowHeigh2"]=true
        dDio["O2_bFollowHeigh3"]=false
      break
      case 3
        dDio["O2_bFollowHeigh1"]=true
        dDio["O2_bFollowHeigh2"]=true
        dDio["O2_bFollowHeigh3"]=false
      break


      case 4
        dDio["O2_bFollowHeigh1"]=false
        dDio["O2_bFollowHeigh2"]=false
        dDio["O2_bFollowHeigh3"]=true
      break
      case 5
        dDio["O2_bFollowHeigh1"]=true
        dDio["O2_bFollowHeigh2"]=false
        dDio["O2_bFollowHeigh3"]=true
      break
      case 6
        dDio["O2_bFollowHeigh1"]=false
        dDio["O2_bFollowHeigh2"]=true
        dDio["O2_bFollowHeigh3"]=true
      break
      case 7,8
        dDio["O2_bFollowHeigh1"]=true
        dDio["O2_bFollowHeigh2"]=true
        dDio["O2_bFollowHeigh3"]=true
      break

    endSwitch


  endIf


end

--- PerforatiAction.pgx ---
public program PerforatiAction(num x_nGasDelay (dimensions=1), num x_nFollowDelay (dimensions=1))
begin

  //穿孔动作
  call KeyDigtalIO(true,true,true,x_nGasDelay,x_nFollowDelay)

end

--- Preset.pgx ---
public program Preset(num& x_nPreset[] (dimensions=2), num x_nIndex (dimensions=1), num x_nPercent (dimensions=1), num x_nHZHight (dimensions=1), num x_nHZLow (dimensions=1))
  local num l_nNum
begin


  //激光工艺设置
  if x_nIndex>0 and x_nIndex<51
    x_nIndex=roundDown(x_nIndex)
    aioSet(aAio["O1_aLasPwr"],x_nPreset[x_nIndex,0]/100*x_nPercent)
    aioSet(aAio["O1_aAirPress"],x_nPreset[x_nIndex,1]/100*x_nPercent)
    //  aioSet(aAio["O1_aFPWM"],x_nPreset[x_nIndex,2]/100*x_nPercent)
    aioSet(aAio["O1_aFPWM"],x_nPreset[x_nIndex,2]*(x_nHZHight-x_nHZLow)/100+x_nHZLow)
    //  aioSet(aAio["O1_aPMW"],x_nPreset[x_nIndex,3]/100*x_nPercent)
    aioSet(aAio["O1_aPMW"],min(max(x_nPreset[x_nIndex,3],0),100))
    aioSet(aAio["O2_aFollowSensitive"],x_nPreset[x_nIndex,4]/100*x_nPercent)
    //  aioSet(aAio["O1_aLasPwr"],x_nPreset[x_nIndex,4])

    if !bDigFollowHight
      return
    endIf
    //2014.05.27
    //对随动高度进行转换
    //0 false false false
    //1~12  true false false
    //13~25  true false false
    //26~38  true false false


    // l_nNum=round(x_nPreset[x_nIndex,4]/12.5)
    l_nNum=round(x_nPreset[x_nIndex,4])
    switch l_nNum
      case 0
        dDio["O2_bFollowHeigh1"]=false
        dDio["O2_bFollowHeigh2"]=false
        dDio["O2_bFollowHeigh3"]=false
      break

      case 1
        dDio["O2_bFollowHeigh1"]=true
        dDio["O2_bFollowHeigh2"]=false
        dDio["O2_bFollowHeigh3"]=false
      break
      case 2
        dDio["O2_bFollowHeigh1"]=false
        dDio["O2_bFollowHeigh2"]=true
        dDio["O2_bFollowHeigh3"]=false
      break
      case 3
        dDio["O2_bFollowHeigh1"]=true
        dDio["O2_bFollowHeigh2"]=true
        dDio["O2_bFollowHeigh3"]=false
      break


      case 4
        dDio["O2_bFollowHeigh1"]=false
        dDio["O2_bFollowHeigh2"]=false
        dDio["O2_bFollowHeigh3"]=true
      break
      case 5
        dDio["O2_bFollowHeigh1"]=true
        dDio["O2_bFollowHeigh2"]=false
        dDio["O2_bFollowHeigh3"]=true
      break
      case 6
        dDio["O2_bFollowHeigh1"]=false
        dDio["O2_bFollowHeigh2"]=true
        dDio["O2_bFollowHeigh3"]=true
      break
      case 7,8
        dDio["O2_bFollowHeigh1"]=true
        dDio["O2_bFollowHeigh2"]=true
        dDio["O2_bFollowHeigh3"]=true
      break

    endSwitch


  endIf


end

--- PresetLaser.pgx ---
public program PresetLaser(num x_nLaserPower (dimensions=1), num x_nPWM (dimensions=1), num x_nPercent (dimensions=1))
  local num l_nNum
begin


  //激光工艺设置
  // if x_nIndex>0 and x_nIndex<51
  // x_nIndex=roundDown(x_nIndex)
  aioSet(aAio["O1_aLasPwr"],min(max(x_nLaserPower,0),100)/100*x_nPercent)
  //  aioSet(aAio["O1_aAirPress"],x_nPreset[x_nIndex,1]/100*x_nPercent)
  //  aioSet(aAio["O1_aFPWM"],x_nPreset[x_nIndex,2]/100*x_nPercent)
  // aioSet(aAio["O1_aFPWM"],x_nPWM*(x_nHZHight-x_nHZLow)/100+x_nHZLow)
  //  aioSet(aAio["O1_aPMW"],x_nPreset[x_nIndex,3]/100*x_nPercent)
  aioSet(aAio["O1_aPMW"],min(max(x_nPWM,0),100))
  // aioSet(aAio["O2_aFollowSensitive"],x_nPreset[x_nIndex,4]/100*x_nPercent)
  //  aioSet(aAio["O1_aLasPwr"],x_nPreset[x_nIndex,4])

  //    if !bDigFollowHight
  //      return
  //    endIf
  //2014.05.27
  //对随动高度进行转换
  //0 false false false
  //1~12  true false false
  //13~25  true false false
  //26~38  true false false


  //    // l_nNum=round(x_nPreset[x_nIndex,4]/12.5)
  //    l_nNum=round(x_nPreset[x_nIndex,4])
  //    switch l_nNum
  //      case 0
  //        dDio["O2_bFollowHeigh1"]=false
  //        dDio["O2_bFollowHeigh2"]=false
  //        dDio["O2_bFollowHeigh3"]=false
  //      break
  //
  //      case 1
  //        dDio["O2_bFollowHeigh1"]=true
  //        dDio["O2_bFollowHeigh2"]=false
  //        dDio["O2_bFollowHeigh3"]=false
  //      break
  //      case 2
  //        dDio["O2_bFollowHeigh1"]=false
  //        dDio["O2_bFollowHeigh2"]=true
  //        dDio["O2_bFollowHeigh3"]=false
  //      break
  //      case 3
  //        dDio["O2_bFollowHeigh1"]=true
  //        dDio["O2_bFollowHeigh2"]=true
  //        dDio["O2_bFollowHeigh3"]=false
  //      break
  //
  //
  //      case 4
  //        dDio["O2_bFollowHeigh1"]=false
  //        dDio["O2_bFollowHeigh2"]=false
  //        dDio["O2_bFollowHeigh3"]=true
  //      break
  //      case 5
  //        dDio["O2_bFollowHeigh1"]=true
  //        dDio["O2_bFollowHeigh2"]=false
  //        dDio["O2_bFollowHeigh3"]=true
  //      break
  //      case 6
  //        dDio["O2_bFollowHeigh1"]=false
  //        dDio["O2_bFollowHeigh2"]=true
  //        dDio["O2_bFollowHeigh3"]=true
  //      break
  //      case 7,8
  //        dDio["O2_bFollowHeigh1"]=true
  //        dDio["O2_bFollowHeigh2"]=true
  //        dDio["O2_bFollowHeigh3"]=true
  //      break
  //
  //    endSwitch
  //

  //  endIf


end

--- ProductPoll.pgx ---
public program ProductPoll(num& x_nCycleCount (dimensions=1), num& x_nInterface (dimensions=1), bool& x_bPause (dimensions=1))
  local string l_sS
begin
  //在生产过程中进行轮询
  //主要是上电，暂停，结束本周期，继续
  //客户可以在这里进行修改




  //上电
  call IOName(1,l_sS)
  if dDio[l_sS]==true
    if !isPowered()
      enablePower()
      logMsg("上电信号被触发")
      if !watch(dDio[l_sS]==false,10)
        disablePower()
        popUpMsg("上电按钮不能超过10秒")
      endIf
    endIf
  endIf

  //结束本周期
  call IOName(5,l_sS)
  if x_nCycleCount!=0 and dDio[l_sS]==true
    delay(0.1)
    if watch(dDio[l_sS]==true,0.1)
      x_nCycleCount=0
    endIf
  endIf



  //立即结束
  call IOName(3,l_sS)
  if dDio[l_sS]==true
    delay(0.05)
    if watch(dDio[l_sS]==true,0.1)

      //2015.01.16立即结束
      aioSet(aAio["Out_a66_81"],0)
      stopMove()

      //
      x_nInterface=9
      logMsg("停止信号被触发")
      return
    endIf
  endIf


  //暂停
  // call IOName(8,l_sS)
  if dDio["In1_bPausCycl"]==true
    if !x_bPause
      // delay(max(0.1,x_nPauseDelay))
      delay(0.05)
      if dDio["In1_bPausCycl"]==true
        logMsg("暂停信号被触发")
        x_bPause=!x_bPause
      endIf
    endIf
    return
  endIf






  //客户可以在这里进行修改 继续按钮
  //继续
  if x_bPause
    //    call IOName(6,l_sS)
    if dDio["In1_bPrdSta1"]==true
      delay(0.1)
      if !watch(dDio["In1_bPrdSta1"]==false,10)
        disablePower()
        popUpMsg("按钮不能超过10秒")
      else
        logMsg("继续信号被触发")
        x_bPause=!x_bPause
      endIf
    endIf
  endIf



end

--- ProductReady.pgx ---
public program ProductReady(num& x_nIndex (dimensions=1), bool x_bFirst (dimensions=1))
  local bool l_bRes
  local num l_nNum
  local string l_sStr
begin



  //2014.05.30
  //工位选择信号
  while true
    //第一工位
    for l_nNum=1 to 4
      if x_bFirst
        l_nNum=1
      endIf
      //测试
      if l_nNum==1 or l_nNum==2
        l_sStr="In1_bPrdSta"+toString("",l_nNum)
      endIf


      //第三工位或者第四工位用户可以进行自定义
      //××××××××××××××××××××××××××××××××××××××××
      if l_nNum==3
        l_sStr="In2_bPrdSta3"
      endIf

      if l_nNum==4
        l_sStr="In2_bPrdSta4"
      endIf
      //×××××××××××××××××××××××××××××××××××××××××
      //信号
      if dDio[l_sStr]==true
        delay(0.1)
        if watch(dDio[l_sStr]==true,0.1)
          logMsg("工位"+toString("",l_nNum)+"信号被触发")
          x_nIndex=l_nNum
          return
        endIf
      endIf

    endFor
    delay(0)
  endWhile



end

--- ReadMe.pgx ---
program ReadMe()
begin
  //与激光相关的内容
  // KeyDigtallO
  //WeldEnd
  //GetKeyIO



  //全局变量说明
  //aAio            全局模拟输出输入变量
  //bAxisDoorEnable 异步轴 安全门打开与关闭
  //bWaitActionOff  在切割点等待输入，如果不满足条件，则关光
  //bWaitFollowDown 等待随动到位信号
  //bWpFinishOut    工位完成，机械手臂到达home点后会发出信号
  //dDio            全局数字输入输出变量
  //sIOName         输入输出名称



  //函数说明
  //








end

--- SafteyIO.pgx ---
public program SafteyIO()
begin
  //对IO做安全化处理
  //报警和下电一般会安全化处理




  //用户自定义IO强制设为0
  //通过变量来设置
  if  bUserIOReset

    if dDio["UsO_bNull5"]==true
      dDio["UsO_bNull5"]=false
      call Digtal2AnalogS(0)
      delay(0.05)
    endIf
  endIf



  call KeyDigtalIO(false,false,false,0,0)

  aioSet(aAio["O1_aLasPwr"],0)
  aioSet(aAio["O1_aAirPress"],0)
  aioSet(aAio["O1_aFPWM"],0)
  aioSet(aAio["O1_aPMW"],0)
  aioSet(aAio["O2_aFollowSensitive"],0)
  dDio["O2_bFollowHeigh1"]=dDio["O2_bFollowHeigh2"]=dDio["O2_bFollowHeigh3"]=false



  //如果是外部轴安全门，下电以后不做动作！
  //2014.06.09
  if bUserIOReset
    //用户自定义IO强制设为0
    if dDio["UsO_bNull4"]==true
      dDio["UsO_bNull4"]=false
      call Digtal2AnalogS(0)
      delay(0.05)
    endIf
    if dDio["UsO_bNull1"]==true or dDio["UsO_bNull2"]==true or dDio["UsO_bNull3"]==true or dDio["UsO_bNull4"]==true or dDio["UsO_bNull5"]==true or dDio["UsO_bNull6"]==true or dDio["UsO_bNull7"]==true or dDio["UsO_bNull8"]==true
      dDio["UsO_bNull1"]=dDio["UsO_bNull2"]=dDio["UsO_bNull3"]=dDio["UsO_bNull4"]=false
      dDio["UsO_bNull5"]=dDio["UsO_bNull6"]=dDio["UsO_bNull7"]=dDio["UsO_bNull8"]=false
      //  dDio["UsO_bNull5"]=dDio["UsO_bNull7"]=dDio["UsO_bNull8"]=false
      call Digtal2AnalogS(0)
      delay(0.05)
      call Digtal2AnalogS(1)

    endIf
  endIf


end

--- SendSpeed.pgx ---
public program SendSpeed(num x_nSpeed (dimensions=1))
begin
  //2014.3.24 设置机器人速度到O2_aNull
  x_nSpeed=max(0,x_nSpeed)
  aioSet(aAio["O2_aNull"],x_nSpeed)



end

--- TrajBypass.pgx ---
public program TrajBypass(bool& x_bByPass (dimensions=1), num x_nIndex (dimensions=1))
begin

  //通过外围信号来对路径是否生产进行判断

  aioSet(aAio["O2_aNull"],x_nIndex)
  logMsg("等待信号"+toString("",x_nIndex)+"路径是否过滤")

  //信号自定义
  //仅仅作为测试使用
  //  wait(aioGet(aAio["In4_a7CurPosH"])==x_nIndex)
  //  x_bByPass=(dDio["In1_bNull1"]==true)

end

--- WaitProIOEnd.pgx ---
public program WaitProIOEnd(num x_nIndex (dimensions=1))
begin
  //等待触发信号初始化
  //在teach库中的product
  switch x_nIndex
    case 1
      wait(dDio["In1_bPrdSta1"]==false)
    break
    case 2
      wait(dDio["In1_bPrdSta2"]==false)
    break

    case 3
      wait(dDio["In2_bPrdSta3"]==false)
    break

    case 4
      wait(dDio["In2_bPrdSta4"]==false)
    break

  endSwitch
end

--- WeldAction.pgx ---
public program WeldAction()
begin

  //焊接收弧点
  dDio["UsO_bNull5"]=true
  // delay(0.005)
  call Digtal2AnalogS(0)



end

--- WeldProgChoose.pgx ---
public program WeldProgChoose(num x_nNum (dimensions=1))
begin

  //激光工序号选择
  //客户自定义
  //2014.2.21  焊接
  //2014.4.15  焊接程序调试

  //强制把收弧点信号置空
  dDio["UsO_bNull5"]=false
  dDio["UsO_bNull4"]=false
  //  if x_nNum!=0
  //    aioSet(aAio["O1_aFPWM"],100)
  //    aioSet(aAio["O1_aPMW"],100)
  //  else
  //
  //
  //  endIf
  aioSet(aAio["O1_aFPWM"],sel(x_nNum==0,0,100))
  aioSet(aAio["O1_aPMW"],sel(x_nNum==0,0,100))
  call Digtal2Analog()
  // delay(0.1)


  //对于值进行解析
  if x_nNum<=0
    dDio["UsO_bNull1"]=dDio["UsO_bNull2"]=dDio["UsO_bNull3"]=false
  else
    dDio["UsO_bNull1"]=(x_nNum%2)==1
    dDio["UsO_bNull2"]=((x_nNum%4)/2>=1)
    dDio["UsO_bNull3"]=(x_nNum>=4)
  endIf

  call Digtal2AnalogS(0)
  if x_nNum!=0
    delay(0.1)
  endIf

end

--- WorkPlaceFinish.pgx ---
public program WorkPlaceFinish(num x_nIndex)
begin
  //2014.05.28
  //工位完成信号
  //x_nIndex 工位1 工位2 工位3 工位4
  //工位完成信号
  //客户可以自己修改
  //在teach库中的product函数中可以看到


  //
  //  if !bWpFinishOut
  //    return
  //  endIf
  //



  //2015.04.20
  //工位完成信号
  if x_nIndex==0
    dDio["O1_bFollowDone"]=true
    call Digtal2Analog()
    delay(1)
    dDio["O1_bFollowDone"]=false
    call Digtal2Analog()
    return
  endIf







  switch x_nIndex
    case 1
      dDio["O2_bSta1Stat"]=true
    break

    case 2
      dDio["O2_bSta2Stat"]=true
    break


    case 3
      dDio["O2_bSta3Stat"]=true
    break

    case 4
      dDio["O2_bSta4Stat"]=true
    break

  endSwitch

  //在低配版本中或者用户自定义中8入8出中可以使用

  switch x_nIndex
    case 1
      dDio["UsO_bNull2"]=true
    break

    case 2
      dDio["UsO_bNull3"]=true
    break


    case 3
      dDio["UsO_bNull4"]=true
    break

    case 4
      dDio["UsO_bNull5"]=true
    break

  endSwitch

  call Digtal2Analog()
  delay(1)

  dDio["O2_bSta1Stat"]=dDio["O2_bSta2Stat"]=dDio["O2_bSta3Stat"]=dDio["O2_bSta4Stat"]=false
  dDio["UsO_bNull2"]=dDio["UsO_bNull3"]=dDio["UsO_bNull4"]=dDio["UsO_bNull5"]=false


  call Digtal2Analog()






end
